Yaskawa INFORM job: pointsmerc3TRJ0.JBI

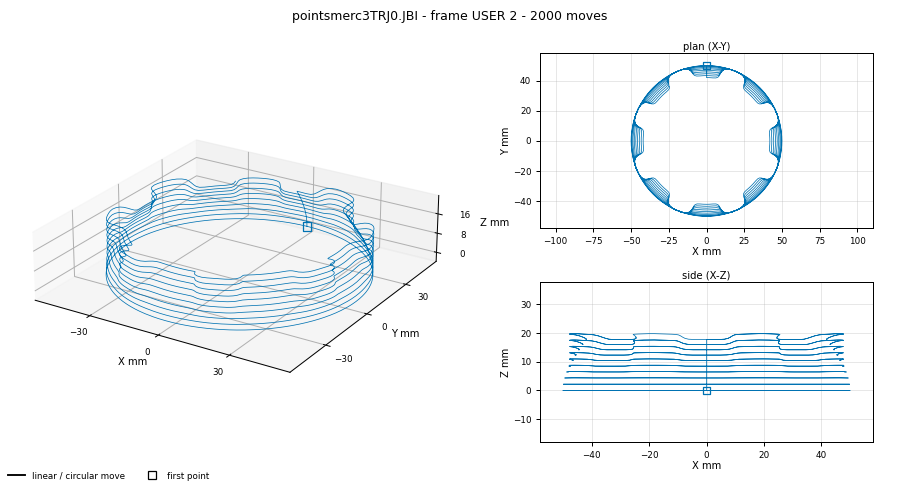
[picture p0: tool path of pointsmerc3TRJ0.JBI in frame USER 2, 2000 of 2000 moves have a stored position in this frame; points joined in program order, loops and branches not executed]
/JOB
//NAME pointsmerc3TRJ0
//POS
///NPOS 2000,0,0,0,0,0
///USER 2
///TOOL 1
///POSTYPE USER
///RECTAN
///RCONF 1,0,0,0,0,0,0,0,0,0,0,0,0,0,0,0,0,0,0,0,0,0,0,0
C00000=0.000,50.000,0.000,-180.0000,0.0000,0.0000
C00001=2.896,49.916,0.000,-180.0000,-0.0000,0.0000
C00002=5.494,49.697,0.000,-180.0000,-0.0000,0.0000
C00003=7.782,49.391,0.000,-180.0000,-0.0000,0.0000
C00004=9.349,49.118,0.000,-180.0000,-0.0000,0.0000
C00005=10.427,48.901,0.000,-180.0000,-0.0000,0.0000
C00006=11.297,48.707,0.000,-180.0000,-0.0000,0.0000
C00007=12.176,48.495,0.000,-180.0000,-0.0000,0.0000
C00008=13.275,48.206,0.000,-180.0000,-0.0000,0.0000
C00009=14.624,47.814,0.000,-180.0000,-0.0000,0.0000
C00010=16.047,47.355,0.000,-180.0000,-0.0000,0.0000
C00011=17.369,46.886,0.000,-180.0000,-0.0000,0.0000
C00012=18.561,46.427,0.000,-180.0000,-0.0000,0.0000
C00013=19.705,45.953,0.000,-180.0000,-0.0000,0.0000
C00014=20.871,45.435,0.000,-180.0000,-0.0000,0.0000
C00015=22.138,44.832,0.000,180.0000,0.0000,0.0000
C00016=23.469,44.150,0.000,180.0000,0.0000,0.0000
C00017=24.700,43.473,0.000,-180.0000,-0.0000,0.0000
C00018=25.682,42.901,0.000,-180.0000,-0.0000,0.0000
C00019=26.453,42.429,0.000,-180.0000,-0.0000,0.0000
C00020=27.205,41.951,0.000,-180.0000,-0.0000,0.0000
C00021=28.121,41.343,0.000,-180.0000,-0.0000,0.0000
C00022=29.422,40.427,0.000,-180.0000,-0.0000,0.0000
C00023=31.256,39.026,0.000,-180.0000,-0.0000,0.0000
C00024=33.248,37.344,0.000,-180.0000,-0.0000,0.0000
C00025=35.355,35.355,0.000,-180.0000,-0.0000,0.0000
C00026=37.344,33.248,0.000,-180.0000,-0.0000,0.0000
C00027=39.026,31.256,0.000,-180.0000,-0.0000,0.0000
C00028=40.427,29.422,0.000,180.0000,0.0000,0.0000
C00029=41.343,28.121,0.000,-180.0000,-0.0000,0.0000
C00030=41.951,27.205,0.000,-180.0000,-0.0000,0.0000
C00031=42.429,26.453,0.000,-180.0000,-0.0000,0.0000
C00032=42.901,25.682,0.000,-180.0000,-0.0000,0.0000
C00033=43.473,24.700,0.000,-180.0000,-0.0000,0.0000
C00034=44.150,23.469,0.000,-180.0000,-0.0000,0.0000
C00035=44.832,22.138,0.000,-180.0000,-0.0000,0.0000
C00036=45.435,20.871,0.000,-180.0000,-0.0000,0.0000
C00037=45.953,19.705,0.000,-180.0000,-0.0000,0.0000
C00038=46.427,18.561,0.000,-180.0000,-0.0000,0.0000
C00039=46.886,17.369,0.000,-180.0000,-0.0000,0.0000
C00040=47.355,16.047,0.000,-180.0000,-0.0000,0.0000
C00041=47.814,14.624,0.000,-180.0000,-0.0000,0.0000
C00042=48.206,13.275,0.000,-180.0000,-0.0000,0.0000
C00043=48.495,12.176,0.000,-180.0000,-0.0000,0.0000
C00044=48.707,11.297,0.000,-180.0000,-0.0000,0.0000
C00045=48.901,10.427,0.000,-180.0000,-0.0000,0.0000
C00046=49.118,9.349,0.000,-180.0000,-0.0000,0.0000
C00047=49.391,7.782,0.000,-180.0000,-0.0000,0.0000
C00048=49.697,5.494,0.000,-180.0000,-0.0000,0.0000
C00049=49.916,2.896,0.000,-180.0000,-0.0000,0.0000
C00050=50.000,0.000,0.000,-180.0000,-0.0000,0.0000
C00051=49.916,-2.896,0.000,180.0000,-0.0000,0.0000
C00052=49.697,-5.494,0.000,180.0000,-0.0000,0.0000
C00053=49.391,-7.782,0.000,180.0000,-0.0000,0.0000
C00054=49.118,-9.349,0.000,180.0000,-0.0000,0.0000
C00055=48.901,-10.427,0.000,180.0000,-0.0000,0.0000
C00056=48.707,-11.297,0.000,180.0000,-0.0000,0.0000
C00057=48.495,-12.176,0.000,180.0000,-0.0000,0.0000
C00058=48.206,-13.275,0.000,180.0000,-0.0000,0.0000
C00059=47.814,-14.624,0.000,180.0000,-0.0000,0.0000
C00060=47.355,-16.047,0.000,180.0000,-0.0000,0.0000
C00061=46.886,-17.369,0.000,180.0000,-0.0000,0.0000
C00062=46.427,-18.561,0.000,180.0000,-0.0000,0.0000
C00063=45.953,-19.705,0.000,180.0000,-0.0000,0.0000
C00064=45.435,-20.871,0.000,180.0000,-0.0000,0.0000
C00065=44.832,-22.138,0.000,180.0000,-0.0000,0.0000
C00066=44.150,-23.469,0.000,180.0000,-0.0000,0.0000
C00067=43.473,-24.700,0.000,180.0000,-0.0000,0.0000
C00068=42.901,-25.682,0.000,180.0000,-0.0000,0.0000
C00069=42.429,-26.453,0.000,180.0000,-0.0000,0.0000
C00070=41.951,-27.205,0.000,180.0000,-0.0000,0.0000
C00071=41.343,-28.121,0.000,180.0000,-0.0000,0.0000
C00072=40.427,-29.422,0.000,180.0000,-0.0000,0.0000
C00073=39.026,-31.256,0.000,180.0000,-0.0000,0.0000
C00074=37.344,-33.248,0.000,180.0000,-0.0000,0.0000
C00075=35.355,-35.355,0.000,180.0000,-0.0000,0.0000
C00076=33.248,-37.344,0.000,180.0000,-0.0000,0.0000
C00077=31.256,-39.026,0.000,180.0000,-0.0000,0.0000
C00078=29.422,-40.427,0.000,180.0000,-0.0000,0.0000
C00079=28.121,-41.343,0.000,180.0000,-0.0000,0.0000
C00080=27.205,-41.951,0.000,180.0000,-0.0000,0.0000
C00081=26.453,-42.429,0.000,180.0000,-0.0000,0.0000
C00082=25.682,-42.901,0.000,180.0000,-0.0000,0.0000
C00083=24.700,-43.473,0.000,-180.0000,0.0000,0.0000
C00084=23.469,-44.150,0.000,180.0000,-0.0000,0.0000
C00085=22.138,-44.832,0.000,180.0000,-0.0000,0.0000
C00086=20.871,-45.435,0.000,180.0000,-0.0000,0.0000
C00087=19.705,-45.953,0.000,180.0000,-0.0000,0.0000
C00088=18.561,-46.427,0.000,180.0000,-0.0000,0.0000
C00089=17.369,-46.886,0.000,180.0000,-0.0000,0.0000
C00090=16.047,-47.355,0.000,180.0000,-0.0000,0.0000
C00091=14.624,-47.814,0.000,180.0000,-0.0000,0.0000
C00092=13.275,-48.206,0.000,180.0000,-0.0000,0.0000
C00093=12.176,-48.495,0.000,180.0000,-0.0000,0.0000
C00094=11.297,-48.707,0.000,180.0000,-0.0000,0.0000
C00095=10.427,-48.901,0.000,180.0000,-0.0000,0.0000
C00096=9.349,-49.118,0.000,180.0000,-0.0000,0.0000
C00097=7.782,-49.391,0.000,180.0000,-0.0000,0.0000
C00098=5.494,-49.697,0.000,180.0000,-0.0000,0.0000
C00099=2.896,-49.916,0.000,180.0000,-0.0000,0.0000
C00100=0.000,-50.000,0.000,-180.0000,-0.0000,0.0000
C00101=0.000,-50.000,0.000,-180.0000,-0.0000,0.0000
C00102=-2.896,-49.916,0.000,-180.0000,-0.0000,0.0000
C00103=-5.494,-49.697,0.000,-180.0000,-0.0000,0.0000
C00104=-7.782,-49.391,0.000,-180.0000,-0.0000,0.0000
C00105=-9.349,-49.118,0.000,-180.0000,-0.0000,0.0000
C00106=-10.427,-48.901,0.000,-180.0000,-0.0000,0.0000
C00107=-11.297,-48.707,0.000,-180.0000,-0.0000,0.0000
C00108=-12.176,-48.495,0.000,-180.0000,-0.0000,0.0000
C00109=-13.275,-48.206,0.000,-180.0000,-0.0000,0.0000
C00110=-14.624,-47.814,0.000,-180.0000,-0.0000,0.0000
C00111=-16.047,-47.355,0.000,-180.0000,-0.0000,0.0000
C00112=-17.369,-46.886,0.000,-180.0000,-0.0000,0.0000
C00113=-18.561,-46.427,0.000,-180.0000,-0.0000,0.0000
C00114=-19.705,-45.953,0.000,-180.0000,-0.0000,0.0000
C00115=-20.871,-45.435,0.000,-180.0000,-0.0000,0.0000
C00116=-22.138,-44.832,0.000,-180.0000,-0.0000,0.0000
C00117=-23.469,-44.150,0.000,-180.0000,-0.0000,0.0000
C00118=-24.700,-43.473,0.000,-180.0000,-0.0000,0.0000
C00119=-25.682,-42.901,0.000,-180.0000,-0.0000,0.0000
C00120=-26.453,-42.429,0.000,-180.0000,-0.0000,0.0000
C00121=-27.205,-41.951,0.000,-180.0000,-0.0000,0.0000
C00122=-28.121,-41.343,0.000,-180.0000,-0.0000,0.0000
C00123=-29.422,-40.427,0.000,-180.0000,-0.0000,0.0000
C00124=-31.256,-39.026,0.000,-180.0000,-0.0000,0.0000
C00125=-33.248,-37.344,0.000,-180.0000,-0.0000,0.0000
C00126=-35.355,-35.355,0.000,-180.0000,-0.0000,0.0000
C00127=-37.344,-33.248,0.000,-180.0000,-0.0000,0.0000
C00128=-39.026,-31.256,0.000,-180.0000,-0.0000,0.0000
C00129=-40.427,-29.422,0.000,-180.0000,-0.0000,0.0000
C00130=-41.343,-28.121,0.000,-180.0000,-0.0000,0.0000
C00131=-41.951,-27.205,0.000,-180.0000,-0.0000,0.0000
C00132=-42.429,-26.453,0.000,-180.0000,-0.0000,0.0000
C00133=-42.901,-25.682,0.000,-180.0000,-0.0000,0.0000
C00134=-43.473,-24.700,0.000,-180.0000,-0.0000,0.0000
C00135=-44.150,-23.469,0.000,-180.0000,-0.0000,0.0000
C00136=-44.832,-22.138,0.000,-180.0000,-0.0000,0.0000
C00137=-45.435,-20.871,0.000,180.0000,0.0000,0.0000
C00138=-45.953,-19.705,0.000,180.0000,0.0000,0.0000
C00139=-46.427,-18.561,0.000,-180.0000,-0.0000,0.0000
C00140=-46.886,-17.369,0.000,-180.0000,-0.0000,0.0000
C00141=-47.355,-16.047,0.000,180.0000,0.0000,0.0000
C00142=-47.814,-14.624,0.000,180.0000,0.0000,0.0000
C00143=-48.206,-13.275,0.000,-180.0000,-0.0000,0.0000
C00144=-48.495,-12.176,0.000,-180.0000,-0.0000,0.0000
C00145=-48.707,-11.297,0.000,-180.0000,-0.0000,0.0000
C00146=-48.901,-10.427,0.000,-180.0000,-0.0000,0.0000
C00147=-49.118,-9.349,0.000,-180.0000,-0.0000,0.0000
C00148=-49.391,-7.782,0.000,-180.0000,-0.0000,0.0000
C00149=-49.697,-5.494,0.000,-180.0000,-0.0000,0.0000
C00150=-49.916,-2.896,0.000,-180.0000,-0.0000,0.0000
C00151=-50.000,0.000,0.000,180.0000,0.0000,0.0000
C00152=-49.916,2.896,0.000,-180.0000,0.0000,0.0000
C00153=-49.697,5.494,0.000,-180.0000,0.0000,0.0000
C00154=-49.391,7.782,0.000,-180.0000,0.0000,0.0000
C00155=-49.118,9.349,0.000,-180.0000,0.0000,0.0000
C00156=-48.901,10.427,0.000,-180.0000,0.0000,0.0000
C00157=-48.707,11.297,0.000,-180.0000,0.0000,0.0000
C00158=-48.495,12.176,0.000,-180.0000,0.0000,0.0000
C00159=-48.206,13.275,0.000,-180.0000,0.0000,0.0000
C00160=-47.814,14.624,0.000,-180.0000,0.0000,0.0000
C00161=-47.355,16.047,0.000,-180.0000,0.0000,0.0000
C00162=-46.886,17.369,0.000,-180.0000,0.0000,0.0000
C00163=-46.427,18.561,0.000,-180.0000,0.0000,0.0000
C00164=-45.953,19.705,0.000,-180.0000,0.0000,0.0000
C00165=-45.435,20.871,0.000,-180.0000,0.0000,0.0000
C00166=-44.832,22.138,0.000,-180.0000,0.0000,0.0000
C00167=-44.150,23.469,0.000,-180.0000,0.0000,0.0000
C00168=-43.473,24.700,0.000,-180.0000,0.0000,0.0000
C00169=-42.901,25.682,0.000,-180.0000,0.0000,0.0000
C00170=-42.429,26.453,0.000,-180.0000,0.0000,0.0000
C00171=-41.951,27.205,0.000,-180.0000,0.0000,0.0000
C00172=-41.343,28.121,0.000,-180.0000,0.0000,0.0000
C00173=-40.427,29.422,0.000,-180.0000,0.0000,0.0000
C00174=-39.026,31.256,0.000,-180.0000,0.0000,0.0000
C00175=-37.344,33.248,0.000,-180.0000,0.0000,0.0000
C00176=-35.355,35.355,0.000,-180.0000,0.0000,0.0000
C00177=-33.248,37.344,0.000,-180.0000,0.0000,0.0000
C00178=-31.256,39.026,0.000,-180.0000,0.0000,0.0000
C00179=-29.422,40.427,0.000,-180.0000,0.0000,0.0000
C00180=-28.121,41.343,0.000,-180.0000,0.0000,0.0000
C00181=-27.205,41.951,0.000,-180.0000,0.0000,0.0000
C00182=-26.453,42.429,0.000,-180.0000,0.0000,0.0000
C00183=-25.682,42.901,0.000,-180.0000,0.0000,0.0000
C00184=-24.700,43.473,0.000,-180.0000,0.0000,0.0000
C00185=-23.469,44.150,0.000,-180.0000,0.0000,0.0000
C00186=-22.138,44.832,0.000,-180.0000,0.0000,0.0000
C00187=-20.871,45.435,0.000,-180.0000,0.0000,0.0000
C00188=-19.705,45.953,0.000,-180.0000,0.0000,0.0000
C00189=-18.561,46.427,0.000,-180.0000,0.0000,0.0000
C00190=-17.369,46.886,0.000,-180.0000,0.0000,0.0000
C00191=-16.047,47.355,0.000,-180.0000,0.0000,0.0000
C00192=-14.624,47.814,0.000,-180.0000,0.0000,0.0000
C00193=-13.275,48.206,0.000,-180.0000,0.0000,0.0000
C00194=-12.176,48.495,0.000,-180.0000,0.0000,0.0000
C00195=-11.297,48.707,0.000,-180.0000,0.0000,0.0000
C00196=-10.427,48.901,0.000,-180.0000,0.0000,0.0000
C00197=-9.349,49.118,0.000,-180.0000,0.0000,0.0000
C00198=-7.782,49.391,0.000,-180.0000,0.0000,0.0000
C00199=-5.494,49.697,0.000,-180.0000,0.0000,0.0000
C00200=-2.896,49.916,0.000,-180.0000,0.0000,0.0000
C00201=0.000,50.000,0.000,-180.0000,0.0000,0.0000
C00202=0.000,49.846,2.195,-172.0982,0.0000,0.0000
C00203=2.882,49.762,2.195,-172.1070,-0.4575,0.0000
C00204=5.471,49.545,2.195,-172.1568,-0.8569,0.0000
C00205=7.753,49.245,2.195,-172.4939,-1.1371,0.0000
C00206=9.315,48.989,2.196,-173.2907,-1.1672,0.0000
C00207=10.389,48.795,2.197,-174.4353,-1.0311,0.0000
C00208=11.257,48.629,2.198,-175.7747,-0.8368,0.0000
C00209=12.134,48.445,2.199,-177.1182,-0.6422,0.0000
C00210=13.230,48.181,2.199,-178.2685,-0.4456,0.0000
C00211=14.582,47.809,2.200,-179.1783,-0.2412,0.0000
C00212=16.014,47.361,2.200,-179.7705,-0.0761,0.0000
C00213=17.348,46.893,2.200,-179.9632,-0.0136,0.0000
C00214=18.554,46.430,2.200,-179.9957,-0.0017,0.0000
C00215=19.712,45.950,2.200,-179.9957,-0.0018,0.0000
C00216=20.891,45.426,2.200,-179.9644,-0.0164,0.0000
C00217=22.166,44.813,2.200,-179.7839,-0.1085,0.0000
C00218=23.495,44.117,2.200,-179.2484,-0.4105,0.0000
C00219=24.714,43.424,2.199,-178.4604,-0.9091,0.0000
C00220=25.676,42.836,2.199,-177.5075,-1.5829,0.0000
C00221=26.426,42.346,2.198,-176.4182,-2.3937,0.0000
C00222=27.157,41.850,2.197,-175.3305,-3.2006,0.0000
C00223=28.054,41.227,2.196,-174.4206,-3.9102,0.0000
C00224=29.339,40.304,2.195,-173.8741,-4.4920,0.0000
C00225=31.165,38.902,2.195,-173.8314,-4.9282,0.0000
C00226=33.149,37.225,2.195,-174.0778,-5.2472,0.0000
C00227=35.246,35.246,2.195,-174.3948,-5.5785,0.0000
C00228=37.225,33.149,2.195,-174.7249,-5.8973,0.0000
C00229=38.902,31.165,2.195,-175.0432,-6.1458,0.0000
C00230=40.304,29.339,2.195,-175.4823,-6.1070,0.0000
C00231=41.227,28.054,2.196,-176.0713,-5.5664,0.0000
C00232=41.850,27.157,2.197,-176.7887,-4.6622,0.0000
C00233=42.346,26.426,2.198,-177.6016,-3.5787,0.0000
C00234=42.836,25.676,2.199,-178.4156,-2.4916,0.0000
C00235=43.424,24.714,2.199,-179.0906,-1.5394,0.0000
C00236=44.117,23.495,2.200,-179.5895,-0.7516,0.0000
C00237=44.813,22.166,2.200,-179.8915,-0.2161,0.0000
C00238=45.426,20.891,2.200,-179.9836,-0.0356,0.0000
C00239=45.950,19.712,2.200,-179.9982,-0.0043,0.0000
C00240=46.430,18.554,2.200,-179.9983,-0.0043,0.0000
C00241=46.893,17.348,2.200,-179.9864,-0.0368,0.0000
C00242=47.361,16.014,2.200,-179.9239,-0.2295,0.0000
C00243=47.809,14.582,2.200,-179.7588,-0.8217,0.0000
C00244=48.181,13.230,2.199,-179.5542,-1.7314,0.0000
C00245=48.445,12.134,2.199,-179.3570,-2.8816,0.0000
C00246=48.629,11.257,2.198,-179.1609,-4.2248,0.0000
C00247=48.795,10.389,2.197,-178.9640,-5.5638,0.0000
C00248=48.989,9.315,2.196,-178.8248,-6.7079,0.0000
C00249=49.245,7.753,2.195,-178.8530,-7.5046,0.0000
C00250=49.545,5.471,2.195,-179.1350,-7.8423,0.0000
C00251=49.762,2.882,2.195,-179.5381,-7.8927,0.0000
C00252=49.846,0.000,2.195,180.0000,-7.9018,0.0000
C00253=49.762,-2.882,2.195,179.5381,-7.8927,0.0000
C00254=49.545,-5.471,2.195,179.1350,-7.8423,0.0000
C00255=49.245,-7.753,2.195,178.8530,-7.5046,0.0000
C00256=48.989,-9.315,2.196,178.8248,-6.7079,0.0000
C00257=48.795,-10.389,2.197,178.9640,-5.5638,0.0000
C00258=48.629,-11.257,2.198,179.1609,-4.2248,0.0000
C00259=48.445,-12.134,2.199,179.3570,-2.8816,0.0000
C00260=48.181,-13.230,2.199,179.5542,-1.7314,0.0000
C00261=47.809,-14.582,2.200,179.7588,-0.8217,0.0000
C00262=47.361,-16.014,2.200,179.9239,-0.2295,0.0000
C00263=46.893,-17.348,2.200,179.9864,-0.0368,0.0000
C00264=46.430,-18.554,2.200,179.9983,-0.0043,0.0000
C00265=45.950,-19.712,2.200,179.9982,-0.0043,0.0000
C00266=45.426,-20.891,2.200,179.9836,-0.0356,0.0000
C00267=44.813,-22.166,2.200,179.8915,-0.2161,0.0000
C00268=44.117,-23.495,2.200,179.5895,-0.7516,0.0000
C00269=43.424,-24.714,2.199,179.0906,-1.5394,0.0000
C00270=42.836,-25.676,2.199,178.4156,-2.4916,0.0000
C00271=42.346,-26.426,2.198,177.6016,-3.5787,0.0000
C00272=41.850,-27.157,2.197,176.7887,-4.6622,0.0000
C00273=41.227,-28.054,2.196,176.0713,-5.5664,0.0000
C00274=40.304,-29.339,2.195,175.4823,-6.1070,0.0000
C00275=38.902,-31.165,2.195,175.0432,-6.1457,0.0000
C00276=37.225,-33.149,2.195,174.7248,-5.8973,0.0000
C00277=35.246,-35.246,2.195,174.3948,-5.5785,0.0000
C00278=33.149,-37.225,2.195,174.0778,-5.2471,0.0000
C00279=31.165,-38.902,2.195,173.8314,-4.9283,0.0000
C00280=29.339,-40.304,2.195,173.8742,-4.4920,0.0000
C00281=28.054,-41.227,2.196,174.4206,-3.9102,0.0000
C00282=27.157,-41.850,2.197,175.3305,-3.2006,0.0000
C00283=26.426,-42.346,2.198,176.4182,-2.3937,0.0000
C00284=25.676,-42.836,2.199,177.5075,-1.5829,0.0000
C00285=24.714,-43.424,2.199,178.4604,-0.9091,0.0000
C00286=23.495,-44.117,2.200,179.2484,-0.4105,0.0000
C00287=22.166,-44.813,2.200,179.7839,-0.1085,0.0000
C00288=20.891,-45.426,2.200,179.9644,-0.0164,0.0000
C00289=19.712,-45.950,2.200,179.9957,-0.0018,0.0000
C00290=18.554,-46.430,2.200,179.9957,-0.0017,0.0000
C00291=17.348,-46.893,2.200,179.9632,-0.0136,0.0000
C00292=16.014,-47.361,2.200,179.7705,-0.0761,0.0000
C00293=14.582,-47.809,2.200,179.1783,-0.2412,0.0000
C00294=13.230,-48.181,2.199,178.2685,-0.4456,0.0000
C00295=12.134,-48.445,2.199,177.1182,-0.6422,0.0000
C00296=11.257,-48.629,2.198,175.7747,-0.8368,0.0000
C00297=10.389,-48.795,2.197,174.4353,-1.0311,0.0000
C00298=9.315,-48.989,2.196,173.2907,-1.1672,0.0000
C00299=7.753,-49.245,2.195,172.4939,-1.1371,0.0000
C00300=5.471,-49.545,2.195,172.1568,-0.8569,0.0000
C00301=2.882,-49.762,2.195,172.1070,-0.4575,0.0000
C00302=0.000,-49.846,2.195,172.0982,0.0000,0.0000
C00303=0.000,-49.846,2.195,172.0982,0.0000,0.0000
C00304=-2.882,-49.762,2.195,172.1071,0.4575,0.0000
C00305=-5.471,-49.545,2.195,172.1568,0.8569,0.0000
C00306=-7.753,-49.245,2.195,172.4939,1.1371,0.0000
C00307=-9.315,-48.989,2.196,173.2907,1.1672,0.0000
C00308=-10.389,-48.795,2.197,174.4353,1.0311,0.0000
C00309=-11.257,-48.629,2.198,175.7747,0.8368,0.0000
C00310=-12.134,-48.445,2.199,177.1182,0.6422,0.0000
C00311=-13.230,-48.181,2.199,178.2685,0.4456,0.0000
C00312=-14.582,-47.809,2.200,179.1783,0.2412,0.0000
C00313=-16.014,-47.361,2.200,179.7705,0.0761,0.0000
C00314=-17.348,-46.893,2.200,179.9632,0.0136,0.0000
C00315=-18.554,-46.430,2.200,179.9957,0.0017,0.0000
C00316=-19.712,-45.950,2.200,179.9957,0.0018,0.0000
C00317=-20.891,-45.426,2.200,179.9644,0.0164,0.0000
C00318=-22.166,-44.813,2.200,179.7839,0.1085,0.0000
C00319=-23.495,-44.117,2.200,179.2484,0.4105,0.0000
C00320=-24.714,-43.424,2.199,178.4604,0.9091,0.0000
C00321=-25.676,-42.836,2.199,177.5075,1.5829,0.0000
C00322=-26.426,-42.346,2.198,176.4182,2.3937,0.0000
C00323=-27.157,-41.850,2.197,175.3305,3.2006,0.0000
C00324=-28.054,-41.227,2.196,174.4206,3.9102,0.0000
C00325=-29.339,-40.304,2.195,173.8741,4.4920,0.0000
C00326=-31.165,-38.902,2.195,173.8314,4.9282,0.0000
C00327=-33.149,-37.225,2.195,174.0778,5.2472,0.0000
C00328=-35.246,-35.246,2.195,174.3948,5.5785,0.0000
C00329=-37.225,-33.149,2.195,174.7249,5.8973,0.0000
C00330=-38.902,-31.165,2.195,175.0432,6.1458,0.0000
C00331=-40.304,-29.339,2.195,175.4823,6.1070,0.0000
C00332=-41.227,-28.054,2.196,176.0713,5.5664,0.0000
C00333=-41.850,-27.157,2.197,176.7887,4.6622,0.0000
C00334=-42.346,-26.426,2.198,177.6016,3.5787,0.0000
C00335=-42.836,-25.676,2.199,178.4156,2.4916,0.0000
C00336=-43.424,-24.714,2.199,179.0906,1.5394,0.0000
C00337=-44.117,-23.495,2.200,179.5895,0.7516,0.0000
C00338=-44.813,-22.166,2.200,179.8915,0.2161,0.0000
C00339=-45.426,-20.891,2.200,179.9836,0.0356,0.0000
C00340=-45.950,-19.712,2.200,179.9982,0.0043,0.0000
C00341=-46.430,-18.554,2.200,179.9983,0.0043,0.0000
C00342=-46.893,-17.348,2.200,179.9864,0.0368,0.0000
C00343=-47.361,-16.014,2.200,179.9239,0.2295,0.0000
C00344=-47.809,-14.582,2.200,179.7588,0.8217,0.0000
C00345=-48.181,-13.230,2.199,179.5542,1.7314,0.0000
C00346=-48.445,-12.134,2.199,179.3570,2.8816,0.0000
C00347=-48.629,-11.257,2.198,179.1609,4.2248,0.0000
C00348=-48.795,-10.389,2.197,178.9640,5.5638,0.0000
C00349=-48.989,-9.315,2.196,178.8248,6.7079,0.0000
C00350=-49.245,-7.753,2.195,178.8530,7.5046,0.0000
C00351=-49.545,-5.471,2.195,179.1350,7.8423,0.0000
C00352=-49.762,-2.882,2.195,179.5381,7.8927,0.0000
C00353=-49.846,0.000,2.195,-180.0000,7.9018,0.0000
C00354=-49.762,2.882,2.195,-179.5381,7.8927,0.0000
C00355=-49.545,5.471,2.195,-179.1350,7.8423,0.0000
C00356=-49.245,7.753,2.195,-178.8530,7.5046,0.0000
C00357=-48.989,9.315,2.196,-178.8248,6.7079,0.0000
C00358=-48.795,10.389,2.197,-178.9640,5.5638,0.0000
C00359=-48.629,11.257,2.198,-179.1609,4.2248,0.0000
C00360=-48.445,12.134,2.199,-179.3570,2.8816,0.0000
C00361=-48.181,13.230,2.199,-179.5542,1.7314,0.0000
C00362=-47.809,14.582,2.200,-179.7588,0.8217,0.0000
C00363=-47.361,16.014,2.200,-179.9239,0.2295,0.0000
C00364=-46.893,17.348,2.200,-179.9864,0.0368,0.0000
C00365=-46.430,18.554,2.200,-179.9983,0.0043,0.0000
C00366=-45.950,19.712,2.200,-179.9982,0.0043,0.0000
C00367=-45.426,20.891,2.200,-179.9836,0.0356,0.0000
C00368=-44.813,22.166,2.200,-179.8915,0.2161,0.0000
C00369=-44.117,23.495,2.200,-179.5895,0.7516,0.0000
C00370=-43.424,24.714,2.199,-179.0906,1.5394,0.0000
C00371=-42.836,25.676,2.199,-178.4156,2.4916,0.0000
C00372=-42.346,26.426,2.198,-177.6016,3.5787,0.0000
C00373=-41.850,27.157,2.197,-176.7887,4.6622,0.0000
C00374=-41.227,28.054,2.196,-176.0713,5.5664,0.0000
C00375=-40.304,29.339,2.195,-175.4823,6.1070,0.0000
C00376=-38.902,31.165,2.195,-175.0432,6.1457,0.0000
C00377=-37.225,33.149,2.195,-174.7248,5.8973,0.0000
C00378=-35.246,35.246,2.195,-174.3948,5.5785,0.0000
C00379=-33.149,37.225,2.195,-174.0778,5.2471,0.0000
C00380=-31.165,38.902,2.195,-173.8314,4.9283,0.0000
C00381=-29.339,40.304,2.195,-173.8742,4.4920,0.0000
C00382=-28.054,41.227,2.196,-174.4206,3.9102,0.0000
C00383=-27.157,41.850,2.197,-175.3305,3.2006,0.0000
C00384=-26.426,42.346,2.198,-176.4182,2.3937,0.0000
C00385=-25.676,42.836,2.199,-177.5075,1.5829,0.0000
C00386=-24.714,43.424,2.199,-178.4604,0.9091,0.0000
C00387=-23.495,44.117,2.200,-179.2484,0.4105,0.0000
C00388=-22.166,44.813,2.200,-179.7839,0.1085,0.0000
C00389=-20.891,45.426,2.200,-179.9644,0.0164,0.0000
C00390=-19.712,45.950,2.200,-179.9957,0.0018,0.0000
C00391=-18.554,46.430,2.200,-179.9957,0.0017,0.0000
C00392=-17.348,46.893,2.200,-179.9632,0.0136,0.0000
C00393=-16.014,47.361,2.200,-179.7705,0.0761,0.0000
C00394=-14.582,47.809,2.200,-179.1783,0.2412,0.0000
C00395=-13.230,48.181,2.199,-178.2685,0.4456,0.0000
C00396=-12.134,48.445,2.199,-177.1182,0.6422,0.0000
C00397=-11.257,48.629,2.198,-175.7747,0.8368,0.0000
C00398=-10.389,48.795,2.197,-174.4353,1.0311,0.0000
C00399=-9.315,48.989,2.196,-173.2907,1.1672,0.0000
C00400=-7.753,49.245,2.195,-172.4939,1.1371,0.0000
C00401=-5.471,49.545,2.195,-172.1568,0.8569,0.0000
C00402=-2.882,49.762,2.195,-172.1071,0.4575,0.0000
C00403=0.000,49.846,2.195,-172.0982,0.0000,0.0000
C00404=0.000,49.410,4.351,-165.2330,0.0000,0.0000
C00405=2.842,49.327,4.351,-165.2490,-0.8462,0.0000
C00406=5.404,49.114,4.351,-165.3368,-1.5509,0.0000
C00407=7.672,48.833,4.355,-165.9287,-1.8917,0.0000
C00408=9.218,48.623,4.363,-167.3753,-1.6057,0.0000
C00409=10.282,48.495,4.374,-169.5506,-1.1016,0.0000
C00410=11.143,48.407,4.384,-172.1383,-0.7944,0.0000
C00411=12.014,48.303,4.391,-174.6908,-0.7528,0.0000
C00412=13.101,48.111,4.395,-176.8484,-0.6476,0.0000
C00413=14.461,47.794,4.396,-178.5414,-0.3774,0.0000
C00414=15.918,47.378,4.398,-179.6165,-0.1196,0.0000
C00415=17.289,46.913,4.399,-179.9364,-0.0233,0.0000
C00416=18.533,46.438,4.400,-179.9926,-0.0029,0.0000
C00417=19.732,45.942,4.400,-179.9927,-0.0031,0.0000
C00418=20.948,45.397,4.399,-179.9386,-0.0286,0.0000
C00419=22.246,44.758,4.398,-179.6442,-0.1866,0.0000
C00420=23.570,44.021,4.396,-178.7016,-0.7644,0.0000
C00421=24.756,43.284,4.395,-177.3126,-1.7696,0.0000
C00422=25.660,42.651,4.391,-175.7085,-3.2179,0.0000
C00423=26.350,42.108,4.384,-173.8623,-4.9857,0.0000
C00424=27.021,41.562,4.374,-171.7926,-6.5822,0.0000
C00425=27.864,40.900,4.363,-169.8688,-7.7398,0.0000
C00426=29.106,39.955,4.355,-168.6177,-8.5390,0.0000
C00427=30.908,38.550,4.351,-168.4253,-9.1948,0.0000
C00428=32.870,36.889,4.351,-168.8566,-9.7634,0.0000
C00429=34.938,34.938,4.351,-169.4418,-10.3834,0.0000
C00430=36.889,32.870,4.351,-170.0527,-10.9799,0.0000
C00431=38.550,30.908,4.351,-170.6177,-11.4240,0.0000
C00432=39.955,29.106,4.355,-171.2923,-11.2544,0.0000
C00433=40.900,27.864,4.363,-172.1392,-10.0380,0.0000
C00434=41.562,27.021,4.374,-173.3503,-8.1529,0.0000
C00435=42.108,26.350,4.384,-174.9857,-6.1144,0.0000
C00436=42.651,25.660,4.391,-176.7731,-4.2848,0.0000
C00437=43.284,24.756,4.395,-178.2285,-2.6861,0.0000
C00438=44.021,23.570,4.396,-179.2354,-1.2982,0.0000
C00439=44.758,22.246,4.398,-179.8134,-0.3558,0.0000
C00440=45.397,20.948,4.399,-179.9714,-0.0614,0.0000
C00441=45.942,19.732,4.400,-179.9969,-0.0073,0.0000
C00442=46.438,18.533,4.400,-179.9971,-0.0074,0.0000
C00443=46.913,17.289,4.399,-179.9767,-0.0636,0.0000
C00444=47.378,15.918,4.398,-179.8804,-0.3835,0.0000
C00445=47.794,14.461,4.396,-179.6224,-1.4586,0.0000
C00446=48.111,13.101,4.395,-179.3514,-3.1514,0.0000
C00447=48.303,12.014,4.391,-179.2440,-5.3088,0.0000
C00448=48.407,11.143,4.384,-179.1981,-7.8609,0.0000
C00449=48.495,10.282,4.374,-178.8799,-10.4474,0.0000
C00450=48.623,9.218,4.363,-178.3546,-12.6196,0.0000
C00451=48.833,7.672,4.355,-178.0498,-14.0635,0.0000
C00452=49.114,5.404,4.351,-178.3969,-14.6577,0.0000
C00453=49.327,2.842,4.351,-179.1250,-14.7494,0.0000
C00454=49.410,0.000,4.351,180.0000,-14.7670,0.0000
C00455=49.327,-2.842,4.351,179.1250,-14.7493,0.0000
C00456=49.114,-5.404,4.351,178.3969,-14.6578,0.0000
C00457=48.833,-7.672,4.355,178.0498,-14.0634,0.0000
C00458=48.623,-9.218,4.363,178.3546,-12.6196,0.0000
C00459=48.495,-10.282,4.374,178.8799,-10.4474,0.0000
C00460=48.407,-11.143,4.384,179.1981,-7.8609,0.0000
C00461=48.303,-12.014,4.391,179.2440,-5.3088,0.0000
C00462=48.111,-13.101,4.395,179.3514,-3.1514,0.0000
C00463=47.794,-14.461,4.396,179.6224,-1.4586,0.0000
C00464=47.378,-15.918,4.398,179.8804,-0.3835,0.0000
C00465=46.913,-17.289,4.399,179.9767,-0.0636,0.0000
C00466=46.438,-18.533,4.400,179.9971,-0.0074,0.0000
C00467=45.942,-19.732,4.400,179.9969,-0.0073,0.0000
C00468=45.397,-20.948,4.399,179.9714,-0.0614,0.0000
C00469=44.758,-22.246,4.398,179.8134,-0.3558,0.0000
C00470=44.021,-23.570,4.396,179.2354,-1.2982,0.0000
C00471=43.284,-24.756,4.395,178.2285,-2.6861,0.0000
C00472=42.651,-25.660,4.391,176.7731,-4.2848,0.0000
C00473=42.108,-26.350,4.384,174.9857,-6.1144,0.0000
C00474=41.562,-27.021,4.374,173.3503,-8.1529,0.0000
C00475=40.900,-27.864,4.363,172.1392,-10.0380,0.0000
C00476=39.955,-29.106,4.355,171.2923,-11.2544,0.0000
C00477=38.550,-30.908,4.351,170.6177,-11.4240,0.0000
C00478=36.889,-32.870,4.351,170.0527,-10.9800,0.0000
C00479=34.938,-34.938,4.351,169.4417,-10.3834,0.0000
C00480=32.870,-36.889,4.351,168.8567,-9.7634,0.0000
C00481=30.908,-38.550,4.351,168.4253,-9.1948,0.0000
C00482=29.106,-39.955,4.355,168.6177,-8.5390,0.0000
C00483=27.864,-40.900,4.363,169.8688,-7.7398,0.0000
C00484=27.021,-41.562,4.374,171.7926,-6.5822,0.0000
C00485=26.350,-42.108,4.384,173.8623,-4.9857,0.0000
C00486=25.660,-42.651,4.391,175.7085,-3.2179,0.0000
C00487=24.756,-43.284,4.395,177.3126,-1.7696,0.0000
C00488=23.570,-44.021,4.396,178.7016,-0.7644,0.0000
C00489=22.246,-44.758,4.398,179.6442,-0.1866,0.0000
C00490=20.948,-45.397,4.399,179.9386,-0.0286,0.0000
C00491=19.732,-45.942,4.400,179.9927,-0.0031,0.0000
C00492=18.533,-46.438,4.400,179.9926,-0.0029,0.0000
C00493=17.289,-46.913,4.399,179.9364,-0.0233,0.0000
C00494=15.918,-47.378,4.398,179.6165,-0.1196,0.0000
C00495=14.461,-47.794,4.396,178.5414,-0.3774,0.0000
C00496=13.101,-48.111,4.395,176.8484,-0.6476,0.0000
C00497=12.014,-48.303,4.391,174.6908,-0.7528,0.0000
C00498=11.143,-48.407,4.384,172.1383,-0.7944,0.0000
C00499=10.282,-48.495,4.374,169.5506,-1.1016,0.0000
C00500=9.218,-48.623,4.363,167.3753,-1.6057,0.0000
C00501=7.672,-48.833,4.355,165.9287,-1.8917,0.0000
C00502=5.404,-49.114,4.351,165.3368,-1.5509,0.0000
C00503=2.842,-49.327,4.351,165.2490,-0.8462,0.0000
C00504=0.000,-49.410,4.351,165.2330,0.0000,0.0000
C00505=0.000,-49.410,4.351,165.2330,0.0000,0.0000
C00506=-2.842,-49.327,4.351,165.2490,0.8461,0.0000
C00507=-5.404,-49.114,4.351,165.3367,1.5509,0.0000
C00508=-7.672,-48.833,4.355,165.9288,1.8917,0.0000
C00509=-9.218,-48.623,4.363,167.3753,1.6057,0.0000
C00510=-10.282,-48.495,4.374,169.5506,1.1016,0.0000
C00511=-11.143,-48.407,4.384,172.1383,0.7944,0.0000
C00512=-12.014,-48.303,4.391,174.6908,0.7528,0.0000
C00513=-13.101,-48.111,4.395,176.8484,0.6476,0.0000
C00514=-14.461,-47.794,4.396,178.5414,0.3774,0.0000
C00515=-15.918,-47.378,4.398,179.6165,0.1196,0.0000
C00516=-17.289,-46.913,4.399,179.9364,0.0233,0.0000
C00517=-18.533,-46.438,4.400,179.9926,0.0029,0.0000
C00518=-19.732,-45.942,4.400,179.9927,0.0031,0.0000
C00519=-20.948,-45.397,4.399,179.9386,0.0286,0.0000
C00520=-22.246,-44.758,4.398,179.6442,0.1866,0.0000
C00521=-23.570,-44.021,4.396,178.7016,0.7644,0.0000
C00522=-24.756,-43.284,4.395,177.3126,1.7696,0.0000
C00523=-25.660,-42.651,4.391,175.7085,3.2179,0.0000
C00524=-26.350,-42.108,4.384,173.8623,4.9857,0.0000
C00525=-27.021,-41.562,4.374,171.7926,6.5822,0.0000
C00526=-27.864,-40.900,4.363,169.8688,7.7398,0.0000
C00527=-29.106,-39.955,4.355,168.6177,8.5390,0.0000
C00528=-30.908,-38.550,4.351,168.4253,9.1948,0.0000
C00529=-32.870,-36.889,4.351,168.8566,9.7634,0.0000
C00530=-34.938,-34.938,4.351,169.4418,10.3834,0.0000
C00531=-36.889,-32.870,4.351,170.0527,10.9799,0.0000
C00532=-38.550,-30.908,4.351,170.6177,11.4240,0.0000
C00533=-39.955,-29.106,4.355,171.2923,11.2544,0.0000
C00534=-40.900,-27.864,4.363,172.1392,10.0380,0.0000
C00535=-41.562,-27.021,4.374,173.3503,8.1529,0.0000
C00536=-42.108,-26.350,4.384,174.9857,6.1144,0.0000
C00537=-42.651,-25.660,4.391,176.7731,4.2848,0.0000
C00538=-43.284,-24.756,4.395,178.2285,2.6861,0.0000
C00539=-44.021,-23.570,4.396,179.2354,1.2982,0.0000
C00540=-44.758,-22.246,4.398,179.8134,0.3558,0.0000
C00541=-45.397,-20.948,4.399,179.9714,0.0614,0.0000
C00542=-45.942,-19.732,4.400,179.9969,0.0073,0.0000
C00543=-46.438,-18.533,4.400,179.9971,0.0074,0.0000
C00544=-46.913,-17.289,4.399,179.9767,0.0636,0.0000
C00545=-47.378,-15.918,4.398,179.8804,0.3835,0.0000
C00546=-47.794,-14.461,4.396,179.6224,1.4586,0.0000
C00547=-48.111,-13.101,4.395,179.3514,3.1514,0.0000
C00548=-48.303,-12.014,4.391,179.2440,5.3088,0.0000
C00549=-48.407,-11.143,4.384,179.1981,7.8609,0.0000
C00550=-48.495,-10.282,4.374,178.8799,10.4474,0.0000
C00551=-48.623,-9.218,4.363,178.3546,12.6196,0.0000
C00552=-48.833,-7.672,4.355,178.0498,14.0635,0.0000
C00553=-49.114,-5.404,4.351,178.3969,14.6577,0.0000
C00554=-49.327,-2.842,4.351,179.1250,14.7494,0.0000
C00555=-49.410,0.000,4.351,-180.0000,14.7670,0.0000
C00556=-49.327,2.842,4.351,-179.1250,14.7493,0.0000
C00557=-49.114,5.404,4.351,-178.3969,14.6578,0.0000
C00558=-48.833,7.672,4.355,-178.0498,14.0634,0.0000
C00559=-48.623,9.218,4.363,-178.3546,12.6196,0.0000
C00560=-48.495,10.282,4.374,-178.8799,10.4474,0.0000
C00561=-48.407,11.143,4.384,-179.1981,7.8609,0.0000
C00562=-48.303,12.014,4.391,-179.2440,5.3088,0.0000
C00563=-48.111,13.101,4.395,-179.3514,3.1514,0.0000
C00564=-47.794,14.461,4.396,-179.6224,1.4586,0.0000
C00565=-47.378,15.918,4.398,-179.8804,0.3835,0.0000
C00566=-46.913,17.289,4.399,-179.9767,0.0636,0.0000
C00567=-46.438,18.533,4.400,-179.9971,0.0074,0.0000
C00568=-45.942,19.732,4.400,-179.9969,0.0073,0.0000
C00569=-45.397,20.948,4.399,-179.9714,0.0614,0.0000
C00570=-44.758,22.246,4.398,-179.8134,0.3558,0.0000
C00571=-44.021,23.570,4.396,-179.2354,1.2982,0.0000
C00572=-43.284,24.756,4.395,-178.2285,2.6861,0.0000
C00573=-42.651,25.660,4.391,-176.7731,4.2848,0.0000
C00574=-42.108,26.350,4.384,-174.9857,6.1144,0.0000
C00575=-41.562,27.021,4.374,-173.3503,8.1529,0.0000
C00576=-40.900,27.864,4.363,-172.1392,10.0380,0.0000
C00577=-39.955,29.106,4.355,-171.2923,11.2544,0.0000
C00578=-38.550,30.908,4.351,-170.6177,11.4240,0.0000
C00579=-36.889,32.870,4.351,-170.0527,10.9800,0.0000
C00580=-34.938,34.938,4.351,-169.4417,10.3834,0.0000
C00581=-32.870,36.889,4.351,-168.8567,9.7634,0.0000
C00582=-30.908,38.550,4.351,-168.4253,9.1948,0.0000
C00583=-29.106,39.955,4.355,-168.6177,8.5390,0.0000
C00584=-27.864,40.900,4.363,-169.8688,7.7398,0.0000
C00585=-27.021,41.562,4.374,-171.7926,6.5822,0.0000
C00586=-26.350,42.108,4.384,-173.8623,4.9857,0.0000
C00587=-25.660,42.651,4.391,-175.7085,3.2179,0.0000
C00588=-24.756,43.284,4.395,-177.3126,1.7696,0.0000
C00589=-23.570,44.021,4.396,-178.7016,0.7644,0.0000
C00590=-22.246,44.758,4.398,-179.6442,0.1866,0.0000
C00591=-20.948,45.397,4.399,-179.9386,0.0286,0.0000
C00592=-19.732,45.942,4.400,-179.9927,0.0031,0.0000
C00593=-18.533,46.438,4.400,-179.9926,0.0029,0.0000
C00594=-17.289,46.913,4.399,-179.9364,0.0233,0.0000
C00595=-15.918,47.378,4.398,-179.6165,0.1196,0.0000
C00596=-14.461,47.794,4.396,-178.5414,0.3774,0.0000
C00597=-13.101,48.111,4.395,-176.8484,0.6476,0.0000
C00598=-12.014,48.303,4.391,-174.6908,0.7528,0.0000
C00599=-11.143,48.407,4.384,-172.1383,0.7944,0.0000
C00600=-10.282,48.495,4.374,-169.5506,1.1016,0.0000
C00601=-9.218,48.623,4.363,-167.3753,1.6057,0.0000
C00602=-7.672,48.833,4.355,-165.9288,1.8917,0.0000
C00603=-5.404,49.114,4.351,-165.3367,1.5509,0.0000
C00604=-2.842,49.327,4.351,-165.2490,0.8461,0.0000
C00605=0.000,49.410,4.351,-165.2330,0.0000,0.0000
C00606=0.000,48.740,6.447,-159.5183,0.0001,0.0000
C00607=2.781,48.660,6.446,-159.5397,-1.1571,0.0000
C00608=5.301,48.453,6.447,-159.6520,-2.0469,0.0000
C00609=7.547,48.199,6.458,-160.4168,-2.1209,0.0000
C00610=9.067,48.057,6.484,-162.4669,-0.9364,0.0000
C00611=10.113,48.028,6.517,-165.7953,0.2947,0.0000
C00612=10.965,48.058,6.549,-169.6341,0.5477,0.0000
C00613=11.826,48.078,6.572,-173.0614,-0.0815,0.0000
C00614=12.898,48.000,6.582,-175.9035,-0.5039,0.0000
C00615=14.270,47.771,6.588,-178.1724,-0.3758,0.0000
C00616=15.768,47.406,6.592,-179.5717,-0.1209,0.0000
C00617=17.193,46.944,6.597,-179.9229,-0.0278,0.0000
C00618=18.501,46.450,6.600,-179.9912,-0.0035,0.0000
C00619=19.763,45.928,6.600,-179.9913,-0.0038,0.0000
C00620=21.037,45.352,6.597,-179.9258,-0.0349,0.0000
C00621=22.372,44.670,6.592,-179.6117,-0.2174,0.0000
C00622=23.689,43.870,6.588,-178.4417,-1.0264,0.0000
C00623=24.821,43.061,6.582,-176.7447,-2.5386,0.0000
C00624=25.634,42.359,6.572,-175.0240,-4.8425,0.0000
C00625=26.229,41.735,6.549,-173.0177,-7.7000,0.0000
C00626=26.810,41.112,6.517,-170.0607,-10.2038,0.0000
C00627=27.570,40.393,6.484,-166.7472,-11.6210,0.0000
C00628=28.746,39.419,6.458,-164.3922,-12.1618,0.0000
C00629=30.513,38.009,6.447,-163.8705,-12.7362,0.0000
C00630=32.441,36.374,6.446,-164.4076,-13.4647,0.0000
C00631=34.464,34.464,6.447,-165.2050,-14.3251,0.0000
C00632=36.374,32.441,6.446,-166.0406,-15.1532,0.0000
C00633=38.009,30.513,6.447,-166.7598,-15.7222,0.0000
C00634=39.419,28.746,6.458,-167.3873,-15.2489,0.0000
C00635=40.393,27.570,6.484,-168.0701,-12.9763,0.0000
C00636=41.112,26.810,6.517,-169.6441,-9.7806,0.0000
C00637=41.735,26.229,6.549,-172.2431,-6.9191,0.0000
C00638=42.359,25.634,6.572,-175.1392,-4.9582,0.0000
C00639=43.061,24.821,6.582,-177.4573,-3.2521,0.0000
C00640=43.870,23.689,6.588,-178.9732,-1.5580,0.0000
C00641=44.670,22.372,6.592,-179.7826,-0.3883,0.0000
C00642=45.352,21.037,6.597,-179.9651,-0.0742,0.0000
C00643=45.928,19.763,6.600,-179.9962,-0.0087,0.0000
C00644=46.450,18.501,6.600,-179.9965,-0.0088,0.0000
C00645=46.944,17.193,6.597,-179.9722,-0.0771,0.0000
C00646=47.406,15.768,6.592,-179.8791,-0.4283,0.0000
C00647=47.771,14.270,6.588,-179.6240,-1.8276,0.0000
C00648=48.000,12.898,6.582,-179.4948,-4.0963,0.0000
C00649=48.078,11.826,6.572,-179.9179,-6.9386,0.0000
C00650=48.058,10.965,6.549,179.4432,-10.3655,0.0000
C00651=48.028,10.113,6.517,179.6960,-14.2045,0.0000
C00652=48.057,9.067,6.484,-179.0180,-17.5307,0.0000
C00653=48.199,7.547,6.458,-177.7490,-19.5693,0.0000
C00654=48.453,5.301,6.447,-177.8170,-20.3344,0.0000
C00655=48.660,2.781,6.446,-178.7651,-20.4559,0.0000
C00656=48.740,0.000,6.447,179.9999,-20.4817,0.0000
C00657=48.660,-2.781,6.446,178.7652,-20.4559,0.0000
C00658=48.453,-5.301,6.447,177.8172,-20.3344,0.0000
C00659=48.199,-7.547,6.458,177.7489,-19.5692,0.0000
C00660=48.057,-9.067,6.484,179.0180,-17.5307,0.0000
C00661=48.028,-10.113,6.517,-179.6960,-14.2045,0.0000
C00662=48.058,-10.965,6.549,-179.4432,-10.3655,0.0000
C00663=48.078,-11.826,6.572,179.9179,-6.9386,0.0000
C00664=48.000,-12.898,6.582,179.4948,-4.0963,0.0000
C00665=47.771,-14.270,6.588,179.6240,-1.8276,0.0000
C00666=47.406,-15.768,6.592,179.8791,-0.4283,0.0000
C00667=46.944,-17.193,6.597,179.9722,-0.0771,0.0000
C00668=46.450,-18.501,6.600,179.9965,-0.0088,0.0000
C00669=45.928,-19.763,6.600,179.9962,-0.0087,0.0000
C00670=45.352,-21.037,6.597,179.9651,-0.0742,0.0000
C00671=44.670,-22.372,6.592,179.7826,-0.3883,0.0000
C00672=43.870,-23.689,6.588,178.9732,-1.5580,0.0000
C00673=43.061,-24.821,6.582,177.4573,-3.2521,0.0000
C00674=42.359,-25.634,6.572,175.1392,-4.9582,0.0000
C00675=41.735,-26.229,6.549,172.2431,-6.9191,0.0000
C00676=41.112,-26.810,6.517,169.6441,-9.7806,0.0000
C00677=40.393,-27.570,6.484,168.0701,-12.9763,0.0000
C00678=39.419,-28.746,6.458,167.3872,-15.2489,0.0000
C00679=38.009,-30.513,6.447,166.7599,-15.7223,0.0000
C00680=36.374,-32.441,6.446,166.0406,-15.1533,0.0000
C00681=34.464,-34.464,6.447,165.2049,-14.3250,0.0000
C00682=32.441,-36.374,6.446,164.4078,-13.4648,0.0000
C00683=30.513,-38.009,6.447,163.8706,-12.7364,0.0000
C00684=28.746,-39.419,6.458,164.3922,-12.1617,0.0000
C00685=27.570,-40.393,6.484,166.7472,-11.6210,0.0000
C00686=26.810,-41.112,6.517,170.0607,-10.2038,0.0000
C00687=26.229,-41.735,6.549,173.0177,-7.7000,0.0000
C00688=25.634,-42.359,6.572,175.0240,-4.8425,0.0000
C00689=24.821,-43.061,6.582,176.7447,-2.5386,0.0000
C00690=23.689,-43.870,6.588,178.4417,-1.0264,0.0000
C00691=22.372,-44.670,6.592,179.6117,-0.2174,0.0000
C00692=21.037,-45.352,6.597,179.9258,-0.0349,0.0000
C00693=19.763,-45.928,6.600,179.9913,-0.0038,0.0000
C00694=18.501,-46.450,6.600,179.9912,-0.0035,0.0000
C00695=17.193,-46.944,6.597,179.9229,-0.0278,0.0000
C00696=15.768,-47.406,6.592,179.5717,-0.1209,0.0000
C00697=14.270,-47.771,6.588,178.1724,-0.3758,0.0000
C00698=12.898,-48.000,6.582,175.9035,-0.5039,0.0000
C00699=11.826,-48.078,6.572,173.0614,-0.0815,0.0000
C00700=10.965,-48.058,6.549,169.6341,0.5477,0.0000
C00701=10.113,-48.028,6.517,165.7953,0.2947,0.0000
C00702=9.067,-48.057,6.484,162.4669,-0.9364,0.0000
C00703=7.547,-48.199,6.458,160.4168,-2.1209,0.0000
C00704=5.301,-48.453,6.447,159.6520,-2.0469,0.0000
C00705=2.781,-48.660,6.446,159.5397,-1.1571,0.0000
C00706=0.000,-48.740,6.447,159.5183,0.0001,0.0000
C00707=0.000,-48.740,6.447,159.5183,0.0001,0.0000
C00708=-2.781,-48.660,6.446,159.5397,1.1569,0.0000
C00709=-5.301,-48.453,6.447,159.6520,2.0467,0.0000
C00710=-7.547,-48.199,6.458,160.4168,2.1210,0.0000
C00711=-9.067,-48.057,6.484,162.4669,0.9364,0.0000
C00712=-10.113,-48.028,6.517,165.7953,-0.2947,0.0000
C00713=-10.965,-48.058,6.549,169.6341,-0.5477,0.0000
C00714=-11.826,-48.078,6.572,173.0614,0.0815,0.0000
C00715=-12.898,-48.000,6.582,175.9035,0.5039,0.0000
C00716=-14.270,-47.771,6.588,178.1724,0.3758,0.0000
C00717=-15.768,-47.406,6.592,179.5717,0.1209,0.0000
C00718=-17.193,-46.944,6.597,179.9229,0.0278,0.0000
C00719=-18.501,-46.450,6.600,179.9912,0.0035,0.0000
C00720=-19.763,-45.928,6.600,179.9913,0.0038,0.0000
C00721=-21.037,-45.352,6.597,179.9258,0.0349,0.0000
C00722=-22.372,-44.670,6.592,179.6117,0.2174,0.0000
C00723=-23.689,-43.870,6.588,178.4417,1.0264,0.0000
C00724=-24.821,-43.061,6.582,176.7447,2.5386,0.0000
C00725=-25.634,-42.359,6.572,175.0240,4.8425,0.0000
C00726=-26.229,-41.735,6.549,173.0177,7.7000,0.0000
C00727=-26.810,-41.112,6.517,170.0607,10.2038,0.0000
C00728=-27.570,-40.393,6.484,166.7472,11.6210,0.0000
C00729=-28.746,-39.419,6.458,164.3922,12.1618,0.0000
C00730=-30.513,-38.009,6.447,163.8705,12.7362,0.0000
C00731=-32.441,-36.374,6.446,164.4076,13.4647,0.0000
C00732=-34.464,-34.464,6.447,165.2050,14.3251,0.0000
C00733=-36.374,-32.441,6.446,166.0406,15.1532,0.0000
C00734=-38.009,-30.513,6.447,166.7598,15.7222,0.0000
C00735=-39.419,-28.746,6.458,167.3873,15.2489,0.0000
C00736=-40.393,-27.570,6.484,168.0701,12.9763,0.0000
C00737=-41.112,-26.810,6.517,169.6441,9.7806,0.0000
C00738=-41.735,-26.229,6.549,172.2431,6.9191,0.0000
C00739=-42.359,-25.634,6.572,175.1392,4.9582,0.0000
C00740=-43.061,-24.821,6.582,177.4573,3.2521,0.0000
C00741=-43.870,-23.689,6.588,178.9732,1.5580,0.0000
C00742=-44.670,-22.372,6.592,179.7826,0.3883,0.0000
C00743=-45.352,-21.037,6.597,179.9651,0.0742,0.0000
C00744=-45.928,-19.763,6.600,179.9962,0.0087,0.0000
C00745=-46.450,-18.501,6.600,179.9965,0.0088,0.0000
C00746=-46.944,-17.193,6.597,179.9722,0.0771,0.0000
C00747=-47.406,-15.768,6.592,179.8791,0.4283,0.0000
C00748=-47.771,-14.270,6.588,179.6240,1.8276,0.0000
C00749=-48.000,-12.898,6.582,179.4948,4.0963,0.0000
C00750=-48.078,-11.826,6.572,179.9179,6.9386,0.0000
C00751=-48.058,-10.965,6.549,-179.4432,10.3655,0.0000
C00752=-48.028,-10.113,6.517,-179.6960,14.2045,0.0000
C00753=-48.057,-9.067,6.484,179.0180,17.5307,0.0000
C00754=-48.199,-7.547,6.458,177.7490,19.5693,0.0000
C00755=-48.453,-5.301,6.447,177.8170,20.3344,0.0000
C00756=-48.660,-2.781,6.446,178.7651,20.4559,0.0000
C00757=-48.740,0.000,6.447,-179.9999,20.4817,0.0000
C00758=-48.660,2.781,6.446,-178.7652,20.4559,0.0000
C00759=-48.453,5.301,6.447,-177.8172,20.3344,0.0000
C00760=-48.199,7.547,6.458,-177.7489,19.5692,0.0000
C00761=-48.057,9.067,6.484,-179.0180,17.5307,0.0000
C00762=-48.028,10.113,6.517,179.6960,14.2045,0.0000
C00763=-48.058,10.965,6.549,179.4432,10.3655,0.0000
C00764=-48.078,11.826,6.572,-179.9179,6.9386,0.0000
C00765=-48.000,12.898,6.582,-179.4948,4.0963,0.0000
C00766=-47.771,14.270,6.588,-179.6240,1.8276,0.0000
C00767=-47.406,15.768,6.592,-179.8791,0.4283,0.0000
C00768=-46.944,17.193,6.597,-179.9722,0.0771,0.0000
C00769=-46.450,18.501,6.600,-179.9965,0.0088,0.0000
C00770=-45.928,19.763,6.600,-179.9962,0.0087,0.0000
C00771=-45.352,21.037,6.597,-179.9651,0.0742,0.0000
C00772=-44.670,22.372,6.592,-179.7826,0.3883,0.0000
C00773=-43.870,23.689,6.588,-178.9732,1.5580,0.0000
C00774=-43.061,24.821,6.582,-177.4573,3.2521,0.0000
C00775=-42.359,25.634,6.572,-175.1392,4.9582,0.0000
C00776=-41.735,26.229,6.549,-172.2431,6.9191,0.0000
C00777=-41.112,26.810,6.517,-169.6441,9.7806,0.0000
C00778=-40.393,27.570,6.484,-168.0701,12.9763,0.0000
C00779=-39.419,28.746,6.458,-167.3872,15.2489,0.0000
C00780=-38.009,30.513,6.447,-166.7599,15.7223,0.0000
C00781=-36.374,32.441,6.446,-166.0406,15.1533,0.0000
C00782=-34.464,34.464,6.447,-165.2049,14.3250,0.0000
C00783=-32.441,36.374,6.446,-164.4078,13.4648,0.0000
C00784=-30.513,38.009,6.447,-163.8706,12.7364,0.0000
C00785=-28.746,39.419,6.458,-164.3922,12.1617,0.0000
C00786=-27.570,40.393,6.484,-166.7472,11.6210,0.0000
C00787=-26.810,41.112,6.517,-170.0607,10.2038,0.0000
C00788=-26.229,41.735,6.549,-173.0177,7.7000,0.0000
C00789=-25.634,42.359,6.572,-175.0240,4.8425,0.0000
C00790=-24.821,43.061,6.582,-176.7447,2.5386,0.0000
C00791=-23.689,43.870,6.588,-178.4417,1.0264,0.0000
C00792=-22.372,44.670,6.592,-179.6117,0.2174,0.0000
C00793=-21.037,45.352,6.597,-179.9258,0.0349,0.0000
C00794=-19.763,45.928,6.600,-179.9913,0.0038,0.0000
C00795=-18.501,46.450,6.600,-179.9912,0.0035,0.0000
C00796=-17.193,46.944,6.597,-179.9229,0.0278,0.0000
C00797=-15.768,47.406,6.592,-179.5717,0.1209,0.0000
C00798=-14.270,47.771,6.588,-178.1724,0.3758,0.0000
C00799=-12.898,48.000,6.582,-175.9035,0.5039,0.0000
C00800=-11.826,48.078,6.572,-173.0614,0.0815,0.0000
C00801=-10.965,48.058,6.549,-169.6341,-0.5477,0.0000
C00802=-10.113,48.028,6.517,-165.7953,-0.2947,0.0000
C00803=-9.067,48.057,6.484,-162.4669,0.9364,0.0000
C00804=-7.547,48.199,6.458,-160.4168,2.1210,0.0000
C00805=-5.301,48.453,6.447,-159.6520,2.0467,0.0000
C00806=-2.781,48.660,6.446,-159.5397,1.1569,0.0000
C00807=0.000,48.740,6.447,-159.5183,0.0001,0.0000
C00808=0.000,47.885,8.473,-154.8794,0.0002,0.0000
C00809=2.703,47.807,8.473,-154.9046,-1.3964,0.0000
C00810=5.169,47.608,8.474,-155.0307,-2.3509,0.0000
C00811=7.387,47.387,8.496,-155.9336,-1.8012,0.0000
C00812=8.874,47.327,8.550,-158.8415,0.9445,0.0000
C00813=9.895,47.421,8.620,-163.9068,3.0310,0.0000
C00814=10.731,47.601,8.688,-169.0791,2.8184,0.0000
C00815=11.577,47.783,8.737,-172.7349,1.1937,0.0000
C00816=12.629,47.854,8.761,-175.6219,-0.0563,0.0000
C00817=14.018,47.741,8.773,-178.1277,-0.2591,0.0000
C00818=15.568,47.442,8.783,-179.6493,-0.0862,0.0000
C00819=17.067,46.986,8.793,-179.9232,-0.0272,0.0000
C00820=18.458,46.467,8.799,-179.9915,-0.0033,0.0000
C00821=19.805,45.909,8.799,-179.9916,-0.0037,0.0000
C00822=21.155,45.292,8.793,-179.9265,-0.0351,0.0000
C00823=22.539,44.555,8.783,-179.6910,-0.1870,0.0000
C00824=23.846,43.670,8.773,-178.4926,-1.1405,0.0000
C00825=24.908,42.767,8.761,-176.8614,-3.0544,0.0000
C00826=25.601,41.974,8.737,-175.6943,-5.9772,0.0000
C00827=26.071,41.247,8.688,-174.2337,-9.7047,0.0000
C00828=26.535,40.528,8.620,-170.6286,-13.4812,0.0000
C00829=27.190,39.740,8.550,-165.3625,-15.4769,0.0000
C00830=28.285,38.731,8.496,-161.2137,-15.4256,0.0000
C00831=30.009,37.319,8.474,-160.1357,-15.6188,0.0000
C00832=31.894,35.716,8.473,-160.6999,-16.4143,0.0000
C00833=33.859,33.859,8.473,-161.6576,-17.4688,0.0000
C00834=35.716,31.894,8.473,-162.6652,-18.4842,0.0000
C00835=37.319,30.009,8.474,-163.4455,-19.1015,0.0000
C00836=38.731,28.285,8.496,-163.7512,-18.0858,0.0000
C00837=39.740,27.190,8.550,-164.0300,-14.0955,0.0000
C00838=40.528,26.535,8.620,-166.3433,-9.1110,0.0000
C00839=41.247,26.071,8.688,-170.2468,-5.6835,0.0000
C00840=41.974,25.601,8.737,-174.0060,-4.2823,0.0000
C00841=42.767,24.908,8.761,-176.9411,-3.1341,0.0000
C00842=43.670,23.846,8.773,-178.8591,-1.5071,0.0000
C00843=44.555,22.539,8.783,-179.8130,-0.3090,0.0000
C00844=45.292,21.155,8.793,-179.9649,-0.0735,0.0000
C00845=45.909,19.805,8.799,-179.9963,-0.0084,0.0000
C00846=46.467,18.458,8.799,-179.9967,-0.0085,0.0000
C00847=46.986,17.067,8.793,-179.9728,-0.0768,0.0000
C00848=47.442,15.568,8.783,-179.9138,-0.3507,0.0000
C00849=47.741,14.018,8.773,-179.7407,-1.8723,0.0000
C00850=47.854,12.629,8.761,-179.9435,-4.3781,0.0000
C00851=47.783,11.577,8.737,178.7966,-7.2635,0.0000
C00852=47.601,10.731,8.688,177.1297,-10.9075,0.0000
C00853=47.421,9.895,8.620,176.8456,-16.0701,0.0000
C00854=47.327,8.874,8.550,178.9873,-21.1555,0.0000
C00855=47.387,7.387,8.496,-178.0274,-24.0538,0.0000
C00856=47.608,5.169,8.474,-177.4070,-24.9468,0.0000
C00857=47.807,2.703,8.473,-178.4581,-25.0874,0.0000
C00858=47.885,0.000,8.473,179.9998,-25.1206,0.0000
C00859=47.807,-2.703,8.473,178.4583,-25.0874,0.0000
C00860=47.608,-5.169,8.474,177.4073,-24.9468,0.0000
C00861=47.387,-7.387,8.496,178.0272,-24.0537,0.0000
C00862=47.327,-8.874,8.550,-178.9873,-21.1555,0.0000
C00863=47.421,-9.895,8.620,-176.8456,-16.0701,0.0000
C00864=47.601,-10.731,8.688,-177.1297,-10.9075,0.0000
C00865=47.783,-11.577,8.737,-178.7966,-7.2635,0.0000
C00866=47.854,-12.629,8.761,179.9435,-4.3781,0.0000
C00867=47.741,-14.018,8.773,179.7407,-1.8723,0.0000
C00868=47.442,-15.568,8.783,179.9138,-0.3507,0.0000
C00869=46.986,-17.067,8.793,179.9728,-0.0768,0.0000
C00870=46.467,-18.458,8.799,179.9967,-0.0085,0.0000
C00871=45.909,-19.805,8.799,179.9963,-0.0084,0.0000
C00872=45.292,-21.155,8.793,179.9649,-0.0735,0.0000
C00873=44.555,-22.539,8.783,179.8130,-0.3090,0.0000
C00874=43.670,-23.846,8.773,178.8591,-1.5071,0.0000
C00875=42.767,-24.908,8.761,176.9411,-3.1341,0.0000
C00876=41.974,-25.601,8.737,174.0060,-4.2823,0.0000
C00877=41.247,-26.071,8.688,170.2468,-5.6835,0.0000
C00878=40.528,-26.535,8.620,166.3433,-9.1110,0.0000
C00879=39.740,-27.190,8.550,164.0300,-14.0955,0.0000
C00880=38.731,-28.285,8.496,163.7510,-18.0857,0.0000
C00881=37.319,-30.009,8.474,163.4457,-19.1017,0.0000
C00882=35.716,-31.894,8.473,162.6653,-18.4844,0.0000
C00883=33.859,-33.859,8.473,161.6573,-17.4685,0.0000
C00884=31.894,-35.716,8.473,160.7001,-16.4145,0.0000
C00885=30.009,-37.319,8.474,160.1359,-15.6190,0.0000
C00886=28.285,-38.731,8.496,161.2136,-15.4254,0.0000
C00887=27.190,-39.740,8.550,165.3625,-15.4769,0.0000
C00888=26.535,-40.528,8.620,170.6286,-13.4812,0.0000
C00889=26.071,-41.247,8.688,174.2337,-9.7047,0.0000
C00890=25.601,-41.974,8.737,175.6943,-5.9772,0.0000
C00891=24.908,-42.767,8.761,176.8614,-3.0544,0.0000
C00892=23.846,-43.670,8.773,178.4926,-1.1405,0.0000
C00893=22.539,-44.555,8.783,179.6910,-0.1870,0.0000
C00894=21.155,-45.292,8.793,179.9265,-0.0351,0.0000
C00895=19.805,-45.909,8.799,179.9916,-0.0037,0.0000
C00896=18.458,-46.467,8.799,179.9915,-0.0033,0.0000
C00897=17.067,-46.986,8.793,179.9232,-0.0272,0.0000
C00898=15.568,-47.442,8.783,179.6493,-0.0862,0.0000
C00899=14.018,-47.741,8.773,178.1277,-0.2591,0.0000
C00900=12.629,-47.854,8.761,175.6219,-0.0563,0.0000
C00901=11.577,-47.783,8.737,172.7349,1.1937,0.0000
C00902=10.731,-47.601,8.688,169.0791,2.8184,0.0000
C00903=9.895,-47.421,8.620,163.9068,3.0310,0.0000
C00904=8.874,-47.327,8.550,158.8415,0.9445,0.0000
C00905=7.387,-47.387,8.496,155.9336,-1.8012,0.0000
C00906=5.169,-47.608,8.474,155.0307,-2.3509,0.0000
C00907=2.703,-47.807,8.473,154.9046,-1.3964,0.0000
C00908=0.000,-47.885,8.473,154.8794,0.0002,0.0000
C00909=0.000,-47.885,8.473,154.8794,0.0002,0.0000
C00910=-2.703,-47.807,8.473,154.9046,1.3962,0.0000
C00911=-5.169,-47.608,8.474,155.0307,2.3506,0.0000
C00912=-7.387,-47.387,8.496,155.9336,1.8014,0.0000
C00913=-8.874,-47.327,8.550,158.8415,-0.9445,0.0000
C00914=-9.895,-47.421,8.620,163.9068,-3.0310,0.0000
C00915=-10.731,-47.601,8.688,169.0791,-2.8184,0.0000
C00916=-11.577,-47.783,8.737,172.7349,-1.1937,0.0000
C00917=-12.629,-47.854,8.761,175.6219,0.0563,0.0000
C00918=-14.018,-47.741,8.773,178.1277,0.2591,0.0000
C00919=-15.568,-47.442,8.783,179.6493,0.0862,0.0000
C00920=-17.067,-46.986,8.793,179.9232,0.0272,0.0000
C00921=-18.458,-46.467,8.799,179.9915,0.0033,0.0000
C00922=-19.805,-45.909,8.799,179.9916,0.0037,0.0000
C00923=-21.155,-45.292,8.793,179.9265,0.0351,0.0000
C00924=-22.539,-44.555,8.783,179.6910,0.1870,0.0000
C00925=-23.846,-43.670,8.773,178.4926,1.1405,0.0000
C00926=-24.908,-42.767,8.761,176.8614,3.0544,0.0000
C00927=-25.601,-41.974,8.737,175.6943,5.9772,0.0000
C00928=-26.071,-41.247,8.688,174.2337,9.7047,0.0000
C00929=-26.535,-40.528,8.620,170.6286,13.4812,0.0000
C00930=-27.190,-39.740,8.550,165.3625,15.4769,0.0000
C00931=-28.285,-38.731,8.496,161.2137,15.4256,0.0000
C00932=-30.009,-37.319,8.474,160.1357,15.6188,0.0000
C00933=-31.894,-35.716,8.473,160.6999,16.4143,0.0000
C00934=-33.859,-33.859,8.473,161.6576,17.4688,0.0000
C00935=-35.716,-31.894,8.473,162.6652,18.4842,0.0000
C00936=-37.319,-30.009,8.474,163.4455,19.1015,0.0000
C00937=-38.731,-28.285,8.496,163.7512,18.0858,0.0000
C00938=-39.740,-27.190,8.550,164.0300,14.0955,0.0000
C00939=-40.528,-26.535,8.620,166.3433,9.1110,0.0000
C00940=-41.247,-26.071,8.688,170.2468,5.6835,0.0000
C00941=-41.974,-25.601,8.737,174.0060,4.2823,0.0000
C00942=-42.767,-24.908,8.761,176.9411,3.1341,0.0000
C00943=-43.670,-23.846,8.773,178.8591,1.5071,0.0000
C00944=-44.555,-22.539,8.783,179.8130,0.3090,0.0000
C00945=-45.292,-21.155,8.793,179.9649,0.0735,0.0000
C00946=-45.909,-19.805,8.799,179.9963,0.0084,0.0000
C00947=-46.467,-18.458,8.799,179.9967,0.0085,0.0000
C00948=-46.986,-17.067,8.793,179.9728,0.0768,0.0000
C00949=-47.442,-15.568,8.783,179.9138,0.3507,0.0000
C00950=-47.741,-14.018,8.773,179.7407,1.8723,0.0000
C00951=-47.854,-12.629,8.761,179.9435,4.3781,0.0000
C00952=-47.783,-11.577,8.737,-178.7966,7.2635,0.0000
C00953=-47.601,-10.731,8.688,-177.1297,10.9075,0.0000
C00954=-47.421,-9.895,8.620,-176.8456,16.0701,0.0000
C00955=-47.327,-8.874,8.550,-178.9873,21.1555,0.0000
C00956=-47.387,-7.387,8.496,178.0274,24.0538,0.0000
C00957=-47.608,-5.169,8.474,177.4070,24.9468,0.0000
C00958=-47.807,-2.703,8.473,178.4581,25.0874,0.0000
C00959=-47.885,0.000,8.473,-179.9998,25.1206,0.0000
C00960=-47.807,2.703,8.473,-178.4583,25.0874,0.0000
C00961=-47.608,5.169,8.474,-177.4073,24.9468,0.0000
C00962=-47.387,7.387,8.496,-178.0272,24.0537,0.0000
C00963=-47.327,8.874,8.550,178.9873,21.1555,0.0000
C00964=-47.421,9.895,8.620,176.8456,16.0701,0.0000
C00965=-47.601,10.731,8.688,177.1297,10.9075,0.0000
C00966=-47.783,11.577,8.737,178.7966,7.2635,0.0000
C00967=-47.854,12.629,8.761,-179.9435,4.3781,0.0000
C00968=-47.741,14.018,8.773,-179.7407,1.8723,0.0000
C00969=-47.442,15.568,8.783,-179.9138,0.3507,0.0000
C00970=-46.986,17.067,8.793,-179.9728,0.0768,0.0000
C00971=-46.467,18.458,8.799,-179.9967,0.0085,0.0000
C00972=-45.909,19.805,8.799,-179.9963,0.0084,0.0000
C00973=-45.292,21.155,8.793,-179.9649,0.0735,0.0000
C00974=-44.555,22.539,8.783,-179.8130,0.3090,0.0000
C00975=-43.670,23.846,8.773,-178.8591,1.5071,0.0000
C00976=-42.767,24.908,8.761,-176.9411,3.1341,0.0000
C00977=-41.974,25.601,8.737,-174.0060,4.2823,0.0000
C00978=-41.247,26.071,8.688,-170.2468,5.6835,0.0000
C00979=-40.528,26.535,8.620,-166.3433,9.1110,0.0000
C00980=-39.740,27.190,8.550,-164.0300,14.0955,0.0000
C00981=-38.731,28.285,8.496,-163.7510,18.0857,0.0000
C00982=-37.319,30.009,8.474,-163.4457,19.1017,0.0000
C00983=-35.716,31.894,8.473,-162.6653,18.4844,0.0000
C00984=-33.859,33.859,8.473,-161.6573,17.4685,0.0000
C00985=-31.894,35.716,8.473,-160.7001,16.4145,0.0000
C00986=-30.009,37.319,8.474,-160.1359,15.6190,0.0000
C00987=-28.285,38.731,8.496,-161.2136,15.4254,0.0000
C00988=-27.190,39.740,8.550,-165.3625,15.4769,0.0000
C00989=-26.535,40.528,8.620,-170.6286,13.4812,0.0000
C00990=-26.071,41.247,8.688,-174.2337,9.7047,0.0000
C00991=-25.601,41.974,8.737,-175.6943,5.9772,0.0000
C00992=-24.908,42.767,8.761,-176.8614,3.0544,0.0000
C00993=-23.846,43.670,8.773,-178.4926,1.1405,0.0000
C00994=-22.539,44.555,8.783,-179.6910,0.1870,0.0000
C00995=-21.155,45.292,8.793,-179.9265,0.0351,0.0000
C00996=-19.805,45.909,8.799,-179.9916,0.0037,0.0000
C00997=-18.458,46.467,8.799,-179.9915,0.0033,0.0000
C00998=-17.067,46.986,8.793,-179.9232,0.0272,0.0000
C00999=-15.568,47.442,8.783,-179.6493,0.0862,0.0000
C01000=-14.018,47.741,8.773,-178.1277,0.2591,0.0000
C01001=-12.629,47.854,8.761,-175.6219,0.0563,0.0000
C01002=-11.577,47.783,8.737,-172.7349,-1.1937,0.0000
C01003=-10.731,47.601,8.688,-169.0791,-2.8184,0.0000
C01004=-9.895,47.421,8.620,-163.9068,-3.0310,0.0000
C01005=-8.874,47.327,8.550,-158.8415,-0.9445,0.0000
C01006=-7.387,47.387,8.496,-155.9336,1.8014,0.0000
C01007=-5.169,47.608,8.474,-155.0307,2.3506,0.0000
C01008=-2.703,47.807,8.473,-154.9046,1.3962,0.0000
C01009=0.000,47.885,8.473,-154.8794,0.0002,0.0000
C01010=0.000,46.884,10.433,-151.1653,0.0002,0.0000
C01011=2.611,46.810,10.432,-151.1930,-1.5762,0.0000
C01012=5.015,46.620,10.433,-151.3262,-2.4871,0.0000
C01013=7.199,46.436,10.471,-152.3977,-0.9762,0.0000
C01014=8.646,46.466,10.562,-156.8195,3.8339,0.0000
C01015=9.635,46.699,10.682,-164.4281,6.1357,0.0000
C01016=10.451,47.054,10.800,-170.7349,4.7296,0.0000
C01017=11.278,47.426,10.887,-173.9779,2.3147,0.0000
C01018=12.303,47.677,10.929,-176.1454,0.4711,0.0000
C01019=13.711,47.704,10.951,-178.4247,-0.0968,0.0000
C01020=15.325,47.486,10.969,-179.8437,-0.0322,0.0000
C01021=16.914,47.036,10.987,-179.9356,-0.0223,0.0000
C01022=18.406,46.487,10.998,-179.9932,-0.0027,0.0000
C01023=19.856,45.886,10.998,-179.9933,-0.0029,0.0000
C01024=21.300,45.220,10.987,-179.9387,-0.0298,0.0000
C01025=22.741,44.414,10.969,-179.8667,-0.0878,0.0000
C01026=24.036,43.427,10.951,-178.8175,-1.0454,0.0000
C01027=25.013,42.412,10.929,-177.6055,-3.0580,0.0000
C01028=25.561,41.510,10.887,-177.3745,-5.8937,0.0000
C01029=25.882,40.662,10.800,-176.7905,-9.8902,0.0000
C01030=26.208,39.834,10.682,-173.2620,-15.3261,0.0000
C01031=26.743,38.970,10.562,-165.8972,-18.9653,0.0000
C01032=27.744,37.925,10.471,-159.0282,-18.3929,0.0000
C01033=29.419,36.512,10.433,-157.1341,-17.9557,0.0000
C01034=31.253,34.946,10.432,-157.6547,-18.7324,0.0000
C01035=33.152,33.152,10.433,-158.7295,-19.9396,0.0000
C01036=34.946,31.253,10.432,-159.8646,-21.1029,0.0000
C01037=36.512,29.419,10.433,-160.6227,-21.6937,0.0000
C01038=37.925,27.744,10.471,-160.3991,-19.8542,0.0000
C01039=38.970,26.743,10.562,-160.4893,-13.3227,0.0000
C01040=39.834,26.208,10.682,-164.5724,-6.4973,0.0000
C01041=40.662,25.882,10.800,-170.0945,-3.1618,0.0000
C01042=41.510,25.561,10.887,-174.1002,-2.6116,0.0000
C01043=42.412,25.013,10.929,-176.9394,-2.3911,0.0000
C01044=43.427,24.036,10.951,-178.9544,-1.1823,0.0000
C01045=44.414,22.741,10.969,-179.9122,-0.1333,0.0000
C01046=45.220,21.300,10.987,-179.9702,-0.0613,0.0000
C01047=45.886,19.856,10.998,-179.9971,-0.0067,0.0000
C01048=46.487,18.406,10.998,-179.9973,-0.0068,0.0000
C01049=47.036,16.914,10.987,-179.9777,-0.0644,0.0000
C01050=47.486,15.325,10.969,-179.9678,-0.1563,0.0000
C01051=47.704,13.711,10.951,-179.9032,-1.5753,0.0000
C01052=47.677,12.303,10.929,179.5279,-3.8544,0.0000
C01053=47.426,11.278,10.887,177.6724,-6.0172,0.0000
C01054=47.054,10.451,10.800,175.2082,-9.2332,0.0000
C01055=46.699,9.635,10.682,173.6324,-15.4805,0.0000
C01056=46.466,8.646,10.562,175.8305,-23.1256,0.0000
C01057=46.436,7.199,10.471,-178.8985,-27.5980,0.0000
C01058=46.620,5.015,10.433,-177.1658,-28.6443,0.0000
C01059=46.810,2.611,10.432,-178.2014,-28.7951,0.0000
C01060=46.884,0.000,10.433,179.9997,-28.8347,0.0000
C01061=46.810,-2.611,10.432,178.2017,-28.7951,0.0000
C01062=46.620,-5.015,10.433,177.1664,-28.6443,0.0000
C01063=46.436,-7.199,10.471,178.8981,-27.5980,0.0000
C01064=46.466,-8.646,10.562,-175.8305,-23.1256,0.0000
C01065=46.699,-9.635,10.682,-173.6324,-15.4805,0.0000
C01066=47.054,-10.451,10.800,-175.2082,-9.2332,0.0000
C01067=47.426,-11.278,10.887,-177.6724,-6.0172,0.0000
C01068=47.677,-12.303,10.929,-179.5279,-3.8544,0.0000
C01069=47.704,-13.711,10.951,179.9032,-1.5753,0.0000
C01070=47.486,-15.325,10.969,179.9678,-0.1563,0.0000
C01071=47.036,-16.914,10.987,179.9777,-0.0644,0.0000
C01072=46.487,-18.406,10.998,179.9973,-0.0068,0.0000
C01073=45.886,-19.856,10.998,179.9971,-0.0067,0.0000
C01074=45.220,-21.300,10.987,179.9702,-0.0613,0.0000
C01075=44.414,-22.741,10.969,179.9122,-0.1333,0.0000
C01076=43.427,-24.036,10.951,178.9544,-1.1823,0.0000
C01077=42.412,-25.013,10.929,176.9394,-2.3911,0.0000
C01078=41.510,-25.561,10.887,174.1002,-2.6116,0.0000
C01079=40.662,-25.882,10.800,170.0945,-3.1618,0.0000
C01080=39.834,-26.208,10.682,164.5724,-6.4973,0.0000
C01081=38.970,-26.743,10.562,160.4893,-13.3227,0.0000
C01082=37.925,-27.744,10.471,160.3988,-19.8540,0.0000
C01083=36.512,-29.419,10.433,160.6231,-21.6940,0.0000
C01084=34.946,-31.253,10.432,159.8649,-21.1031,0.0000
C01085=33.152,-33.152,10.433,158.7292,-19.9393,0.0000
C01086=31.253,-34.946,10.432,157.6550,-18.7327,0.0000
C01087=29.419,-36.512,10.433,157.1345,-17.9561,0.0000
C01088=27.744,-37.925,10.471,159.0280,-18.3926,0.0000
C01089=26.743,-38.970,10.562,165.8972,-18.9653,0.0000
C01090=26.208,-39.834,10.682,173.2620,-15.3261,0.0000
C01091=25.882,-40.662,10.800,176.7905,-9.8902,0.0000
C01092=25.561,-41.510,10.887,177.3745,-5.8937,0.0000
C01093=25.013,-42.412,10.929,177.6055,-3.0580,0.0000
C01094=24.036,-43.427,10.951,178.8175,-1.0454,0.0000
C01095=22.741,-44.414,10.969,179.8667,-0.0878,0.0000
C01096=21.300,-45.220,10.987,179.9387,-0.0298,0.0000
C01097=19.856,-45.886,10.998,179.9933,-0.0029,0.0000
C01098=18.406,-46.487,10.998,179.9932,-0.0027,0.0000
C01099=16.914,-47.036,10.987,179.9356,-0.0223,0.0000
C01100=15.325,-47.486,10.969,179.8437,-0.0322,0.0000
C01101=13.711,-47.704,10.951,178.4247,-0.0968,0.0000
C01102=12.303,-47.677,10.929,176.1454,0.4711,0.0000
C01103=11.278,-47.426,10.887,173.9779,2.3147,0.0000
C01104=10.451,-47.054,10.800,170.7349,4.7296,0.0000
C01105=9.635,-46.699,10.682,164.4281,6.1357,0.0000
C01106=8.646,-46.466,10.562,156.8195,3.8339,0.0000
C01107=7.199,-46.436,10.471,152.3977,-0.9762,0.0000
C01108=5.015,-46.620,10.433,151.3262,-2.4871,0.0000
C01109=2.611,-46.810,10.432,151.1930,-1.5762,0.0000
C01110=0.000,-46.884,10.433,151.1653,0.0002,0.0000
C01111=0.000,-46.884,10.433,151.1653,0.0002,0.0000
C01112=-2.611,-46.810,10.432,151.1930,1.5758,0.0000
C01113=-5.015,-46.620,10.433,151.3262,2.4866,0.0000
C01114=-7.199,-46.436,10.471,152.3977,0.9765,0.0000
C01115=-8.646,-46.466,10.562,156.8195,-3.8339,0.0000
C01116=-9.635,-46.699,10.682,164.4281,-6.1357,0.0000
C01117=-10.451,-47.054,10.800,170.7349,-4.7296,0.0000
C01118=-11.278,-47.426,10.887,173.9779,-2.3147,0.0000
C01119=-12.303,-47.677,10.929,176.1454,-0.4711,0.0000
C01120=-13.711,-47.704,10.951,178.4247,0.0968,0.0000
C01121=-15.325,-47.486,10.969,179.8437,0.0322,0.0000
C01122=-16.914,-47.036,10.987,179.9356,0.0223,0.0000
C01123=-18.406,-46.487,10.998,179.9932,0.0027,0.0000
C01124=-19.856,-45.886,10.998,179.9933,0.0029,0.0000
C01125=-21.300,-45.220,10.987,179.9387,0.0298,0.0000
C01126=-22.741,-44.414,10.969,179.8667,0.0878,0.0000
C01127=-24.036,-43.427,10.951,178.8175,1.0454,0.0000
C01128=-25.013,-42.412,10.929,177.6055,3.0580,0.0000
C01129=-25.561,-41.510,10.887,177.3745,5.8937,0.0000
C01130=-25.882,-40.662,10.800,176.7905,9.8902,0.0000
C01131=-26.208,-39.834,10.682,173.2620,15.3261,0.0000
C01132=-26.743,-38.970,10.562,165.8972,18.9653,0.0000
C01133=-27.744,-37.925,10.471,159.0282,18.3929,0.0000
C01134=-29.419,-36.512,10.433,157.1341,17.9557,0.0000
C01135=-31.253,-34.946,10.432,157.6547,18.7324,0.0000
C01136=-33.152,-33.152,10.433,158.7295,19.9396,0.0000
C01137=-34.946,-31.253,10.432,159.8646,21.1029,0.0000
C01138=-36.512,-29.419,10.433,160.6227,21.6937,0.0000
C01139=-37.925,-27.744,10.471,160.3991,19.8542,0.0000
C01140=-38.970,-26.743,10.562,160.4893,13.3227,0.0000
C01141=-39.834,-26.208,10.682,164.5724,6.4973,0.0000
C01142=-40.662,-25.882,10.800,170.0945,3.1618,0.0000
C01143=-41.510,-25.561,10.887,174.1002,2.6116,0.0000
C01144=-42.412,-25.013,10.929,176.9394,2.3911,0.0000
C01145=-43.427,-24.036,10.951,178.9544,1.1823,0.0000
C01146=-44.414,-22.741,10.969,179.9122,0.1333,0.0000
C01147=-45.220,-21.300,10.987,179.9702,0.0613,0.0000
C01148=-45.886,-19.856,10.998,179.9971,0.0067,0.0000
C01149=-46.487,-18.406,10.998,179.9973,0.0068,0.0000
C01150=-47.036,-16.914,10.987,179.9777,0.0644,0.0000
C01151=-47.486,-15.325,10.969,179.9678,0.1563,0.0000
C01152=-47.704,-13.711,10.951,179.9032,1.5753,0.0000
C01153=-47.677,-12.303,10.929,-179.5279,3.8544,0.0000
C01154=-47.426,-11.278,10.887,-177.6724,6.0172,0.0000
C01155=-47.054,-10.451,10.800,-175.2082,9.2332,0.0000
C01156=-46.699,-9.635,10.682,-173.6324,15.4805,0.0000
C01157=-46.466,-8.646,10.562,-175.8305,23.1256,0.0000
C01158=-46.436,-7.199,10.471,178.8985,27.5980,0.0000
C01159=-46.620,-5.015,10.433,177.1658,28.6443,0.0000
C01160=-46.810,-2.611,10.432,178.2014,28.7951,0.0000
C01161=-46.884,0.000,10.433,-179.9997,28.8347,0.0000
C01162=-46.810,2.611,10.432,-178.2017,28.7951,0.0000
C01163=-46.620,5.015,10.433,-177.1664,28.6443,0.0000
C01164=-46.436,7.199,10.471,-178.8981,27.5980,0.0000
C01165=-46.466,8.646,10.562,175.8305,23.1256,0.0000
C01166=-46.699,9.635,10.682,173.6324,15.4805,0.0000
C01167=-47.054,10.451,10.800,175.2082,9.2332,0.0000
C01168=-47.426,11.278,10.887,177.6724,6.0172,0.0000
C01169=-47.677,12.303,10.929,179.5279,3.8544,0.0000
C01170=-47.704,13.711,10.951,-179.9032,1.5753,0.0000
C01171=-47.486,15.325,10.969,-179.9678,0.1563,0.0000
C01172=-47.036,16.914,10.987,-179.9777,0.0644,0.0000
C01173=-46.487,18.406,10.998,-179.9973,0.0068,0.0000
C01174=-45.886,19.856,10.998,-179.9971,0.0067,0.0000
C01175=-45.220,21.300,10.987,-179.9702,0.0613,0.0000
C01176=-44.414,22.741,10.969,-179.9122,0.1333,0.0000
C01177=-43.427,24.036,10.951,-178.9544,1.1823,0.0000
C01178=-42.412,25.013,10.929,-176.9394,2.3911,0.0000
C01179=-41.510,25.561,10.887,-174.1002,2.6116,0.0000
C01180=-40.662,25.882,10.800,-170.0945,3.1618,0.0000
C01181=-39.834,26.208,10.682,-164.5724,6.4973,0.0000
C01182=-38.970,26.743,10.562,-160.4893,13.3227,0.0000
C01183=-37.925,27.744,10.471,-160.3988,19.8540,0.0000
C01184=-36.512,29.419,10.433,-160.6231,21.6940,0.0000
C01185=-34.946,31.253,10.432,-159.8649,21.1031,0.0000
C01186=-33.152,33.152,10.433,-158.7292,19.9393,0.0000
C01187=-31.253,34.946,10.432,-157.6550,18.7327,0.0000
C01188=-29.419,36.512,10.433,-157.1345,17.9561,0.0000
C01189=-27.744,37.925,10.471,-159.0280,18.3926,0.0000
C01190=-26.743,38.970,10.562,-165.8972,18.9653,0.0000
C01191=-26.208,39.834,10.682,-173.2620,15.3261,0.0000
C01192=-25.882,40.662,10.800,-176.7905,9.8902,0.0000
C01193=-25.561,41.510,10.887,-177.3745,5.8937,0.0000
C01194=-25.013,42.412,10.929,-177.6055,3.0580,0.0000
C01195=-24.036,43.427,10.951,-178.8175,1.0454,0.0000
C01196=-22.741,44.414,10.969,-179.8667,0.0878,0.0000
C01197=-21.300,45.220,10.987,-179.9387,0.0298,0.0000
C01198=-19.856,45.886,10.998,-179.9933,0.0029,0.0000
C01199=-18.406,46.487,10.998,-179.9932,0.0027,0.0000
C01200=-16.914,47.036,10.987,-179.9356,0.0223,0.0000
C01201=-15.325,47.486,10.969,-179.8437,0.0322,0.0000
C01202=-13.711,47.704,10.951,-178.4247,0.0968,0.0000
C01203=-12.303,47.677,10.929,-176.1454,-0.4711,0.0000
C01204=-11.278,47.426,10.887,-173.9779,-2.3147,0.0000
C01205=-10.451,47.054,10.800,-170.7349,-4.7296,0.0000
C01206=-9.635,46.699,10.682,-164.4281,-6.1357,0.0000
C01207=-8.646,46.466,10.562,-156.8195,-3.8339,0.0000
C01208=-7.199,46.436,10.471,-152.3977,0.9765,0.0000
C01209=-5.015,46.620,10.433,-151.3262,2.4866,0.0000
C01210=-2.611,46.810,10.432,-151.1930,1.5758,0.0000
C01211=0.000,46.884,10.433,-151.1653,0.0002,0.0000
C01212=0.000,45.772,12.331,-148.2173,0.0003,0.0000
C01213=2.510,45.702,12.329,-148.2466,-1.7081,0.0000
C01214=4.844,45.521,12.332,-148.3842,-2.4822,0.0000
C01215=6.990,45.375,12.387,-149.7196,0.2799,0.0000
C01216=8.390,45.503,12.523,-156.6479,7.2043,0.0000
C01217=9.343,45.885,12.705,-167.0222,8.2576,0.0000
C01218=10.132,46.432,12.887,-173.6461,5.1271,0.0000
C01219=10.935,47.018,13.022,-176.2893,2.4011,0.0000
C01220=11.930,47.474,13.088,-177.4312,0.7183,0.0000
C01221=13.360,47.661,13.123,-179.0290,0.0208,0.0000
C01222=15.047,47.537,13.151,179.8657,0.0220,0.0000
C01223=16.738,47.094,13.179,-179.9573,-0.0145,0.0000
C01224=18.347,46.510,13.197,-179.9960,-0.0016,0.0000
C01225=19.915,45.860,13.197,-179.9960,-0.0018,0.0000
C01226=21.465,45.136,13.179,-179.9596,-0.0199,0.0000
C01227=22.974,44.253,13.151,179.8895,0.0794,0.0000
C01228=24.255,43.149,13.123,-179.3281,-0.7013,0.0000
C01229=25.133,42.005,13.088,-178.6911,-2.3242,0.0000
C01230=25.514,40.979,13.022,-179.0750,-4.3212,0.0000
C01231=25.668,39.997,12.887,-179.1463,-8.1134,0.0000
C01232=25.839,39.052,12.705,-176.7006,-14.9934,0.0000
C01233=26.243,38.108,12.523,-168.2536,-21.5152,0.0000
C01234=27.143,37.028,12.387,-157.7615,-21.0999,0.0000
C01235=28.763,35.614,12.332,-154.7665,-19.8591,0.0000
C01236=30.541,34.091,12.329,-155.1829,-20.5413,0.0000
C01237=32.366,32.366,12.331,-156.3406,-21.8659,0.0000
C01238=34.091,30.541,12.329,-157.5673,-23.1433,0.0000
C01239=35.614,28.763,12.332,-158.2333,-23.6374,0.0000
C01240=37.028,27.143,12.387,-157.3703,-20.6767,0.0000
C01241=38.108,26.243,12.523,-158.0679,-10.9174,0.0000
C01242=39.052,25.839,12.705,-164.9828,-3.1869,0.0000
C01243=39.997,25.668,12.887,-171.8857,-0.8452,0.0000
C01244=40.979,25.514,13.022,-175.6783,-0.9224,0.0000
C01245=42.005,25.133,13.088,-177.6752,-1.3079,0.0000
C01246=43.149,24.255,13.123,-179.2987,-0.6719,0.0000
C01247=44.253,22.974,13.151,179.9206,0.1105,0.0000
C01248=45.136,21.465,13.179,-179.9801,-0.0404,0.0000
C01249=45.860,19.915,13.197,-179.9982,-0.0040,0.0000
C01250=46.510,18.347,13.197,-179.9984,-0.0040,0.0000
C01251=47.094,16.738,13.179,-179.9855,-0.0427,0.0000
C01252=47.537,15.047,13.151,179.9780,0.1343,0.0000
C01253=47.661,13.360,13.123,179.9792,-0.9710,0.0000
C01254=47.474,11.930,13.088,179.2810,-2.5686,0.0000
C01255=47.018,10.935,13.022,177.5938,-3.7074,0.0000
C01256=46.432,10.132,12.887,174.8414,-6.3283,0.0000
C01257=45.885,9.343,12.705,171.5291,-12.8409,0.0000
C01258=45.503,8.390,12.523,172.1606,-23.1570,0.0000
C01259=45.375,6.990,12.387,179.6759,-30.2800,0.0000
C01260=45.521,4.844,12.332,-177.0859,-31.5827,0.0000
C01261=45.702,2.510,12.329,-177.9915,-31.7377,0.0000
C01262=45.772,0.000,12.331,179.9996,-31.7827,0.0000
C01263=45.702,-2.510,12.329,177.9919,-31.7377,0.0000
C01264=45.521,-4.844,12.332,177.0867,-31.5827,0.0000
C01265=45.375,-6.990,12.387,-179.6765,-30.2800,0.0000
C01266=45.503,-8.390,12.523,-172.1606,-23.1570,0.0000
C01267=45.885,-9.343,12.705,-171.5291,-12.8409,0.0000
C01268=46.432,-10.132,12.887,-174.8414,-6.3283,0.0000
C01269=47.018,-10.935,13.022,-177.5938,-3.7074,0.0000
C01270=47.474,-11.930,13.088,-179.2810,-2.5686,0.0000
C01271=47.661,-13.360,13.123,-179.9792,-0.9710,0.0000
C01272=47.537,-15.047,13.151,-179.9780,0.1343,0.0000
C01273=47.094,-16.738,13.179,179.9855,-0.0427,0.0000
C01274=46.510,-18.347,13.197,179.9984,-0.0040,0.0000
C01275=45.860,-19.915,13.197,179.9982,-0.0040,0.0000
C01276=45.136,-21.465,13.179,179.9801,-0.0404,0.0000
C01277=44.253,-22.974,13.151,-179.9206,0.1105,0.0000
C01278=43.149,-24.255,13.123,179.2987,-0.6719,0.0000
C01279=42.005,-25.133,13.088,177.6752,-1.3079,0.0000
C01280=40.979,-25.514,13.022,175.6783,-0.9224,0.0000
C01281=39.997,-25.668,12.887,171.8857,-0.8452,0.0000
C01282=39.052,-25.839,12.705,164.9828,-3.1869,0.0000
C01283=38.108,-26.243,12.523,158.0679,-10.9174,0.0000
C01284=37.028,-27.143,12.387,157.3700,-20.6763,0.0000
C01285=35.614,-28.763,12.332,158.2337,-23.6380,0.0000
C01286=34.091,-30.541,12.329,157.5676,-23.1436,0.0000
C01287=32.366,-32.366,12.331,156.3402,-21.8655,0.0000
C01288=30.541,-34.091,12.329,155.1831,-20.5417,0.0000
C01289=28.763,-35.614,12.332,154.7670,-19.8596,0.0000
C01290=27.143,-37.028,12.387,157.7612,-21.0996,0.0000
C01291=26.243,-38.108,12.523,168.2536,-21.5152,0.0000
C01292=25.839,-39.052,12.705,176.7006,-14.9934,0.0000
C01293=25.668,-39.997,12.887,179.1463,-8.1134,0.0000
C01294=25.514,-40.979,13.022,179.0750,-4.3212,0.0000
C01295=25.133,-42.005,13.088,178.6911,-2.3242,0.0000
C01296=24.255,-43.149,13.123,179.3281,-0.7013,0.0000
C01297=22.974,-44.253,13.151,-179.8895,0.0794,0.0000
C01298=21.465,-45.136,13.179,179.9596,-0.0199,0.0000
C01299=19.915,-45.860,13.197,179.9960,-0.0018,0.0000
C01300=18.347,-46.510,13.197,179.9960,-0.0016,0.0000
C01301=16.738,-47.094,13.179,179.9573,-0.0145,0.0000
C01302=15.047,-47.537,13.151,-179.8657,0.0220,0.0000
C01303=13.360,-47.661,13.123,179.0290,0.0208,0.0000
C01304=11.930,-47.474,13.088,177.4312,0.7183,0.0000
C01305=10.935,-47.018,13.022,176.2893,2.4011,0.0000
C01306=10.132,-46.432,12.887,173.6461,5.1271,0.0000
C01307=9.343,-45.885,12.705,167.0222,8.2576,0.0000
C01308=8.390,-45.503,12.523,156.6479,7.2043,0.0000
C01309=6.990,-45.375,12.387,149.7196,0.2799,0.0000
C01310=4.844,-45.521,12.332,148.3842,-2.4822,0.0000
C01311=2.510,-45.702,12.329,148.2466,-1.7081,0.0000
C01312=0.000,-45.772,12.331,148.2173,0.0003,0.0000
C01313=0.000,-45.772,12.331,148.2173,0.0003,0.0000
C01314=-2.510,-45.702,12.329,148.2466,1.7077,0.0000
C01315=-4.844,-45.521,12.332,148.3843,2.4815,0.0000
C01316=-6.990,-45.375,12.387,149.7196,-0.2794,0.0000
C01317=-8.390,-45.503,12.523,156.6479,-7.2043,0.0000
C01318=-9.343,-45.885,12.705,167.0222,-8.2576,0.0000
C01319=-10.132,-46.432,12.887,173.6461,-5.1271,0.0000
C01320=-10.935,-47.018,13.022,176.2893,-2.4011,0.0000
C01321=-11.930,-47.474,13.088,177.4312,-0.7183,0.0000
C01322=-13.360,-47.661,13.123,179.0290,-0.0208,0.0000
C01323=-15.047,-47.537,13.151,-179.8657,-0.0220,0.0000
C01324=-16.738,-47.094,13.179,179.9573,0.0145,0.0000
C01325=-18.347,-46.510,13.197,179.9960,0.0016,0.0000
C01326=-19.915,-45.860,13.197,179.9960,0.0018,0.0000
C01327=-21.465,-45.136,13.179,179.9596,0.0199,0.0000
C01328=-22.974,-44.253,13.151,-179.8895,-0.0794,0.0000
C01329=-24.255,-43.149,13.123,179.3281,0.7013,0.0000
C01330=-25.133,-42.005,13.088,178.6911,2.3242,0.0000
C01331=-25.514,-40.979,13.022,179.0750,4.3212,0.0000
C01332=-25.668,-39.997,12.887,179.1463,8.1134,0.0000
C01333=-25.839,-39.052,12.705,176.7006,14.9934,0.0000
C01334=-26.243,-38.108,12.523,168.2536,21.5152,0.0000
C01335=-27.143,-37.028,12.387,157.7615,21.0999,0.0000
C01336=-28.763,-35.614,12.332,154.7665,19.8591,0.0000
C01337=-30.541,-34.091,12.329,155.1829,20.5413,0.0000
C01338=-32.366,-32.366,12.331,156.3406,21.8659,0.0000
C01339=-34.091,-30.541,12.329,157.5673,23.1433,0.0000
C01340=-35.614,-28.763,12.332,158.2333,23.6374,0.0000
C01341=-37.028,-27.143,12.387,157.3703,20.6767,0.0000
C01342=-38.108,-26.243,12.523,158.0679,10.9174,0.0000
C01343=-39.052,-25.839,12.705,164.9828,3.1869,0.0000
C01344=-39.997,-25.668,12.887,171.8857,0.8452,0.0000
C01345=-40.979,-25.514,13.022,175.6783,0.9224,0.0000
C01346=-42.005,-25.133,13.088,177.6752,1.3079,0.0000
C01347=-43.149,-24.255,13.123,179.2987,0.6719,0.0000
C01348=-44.253,-22.974,13.151,-179.9206,-0.1105,0.0000
C01349=-45.136,-21.465,13.179,179.9801,0.0404,0.0000
C01350=-45.860,-19.915,13.197,179.9982,0.0040,0.0000
C01351=-46.510,-18.347,13.197,179.9984,0.0040,0.0000
C01352=-47.094,-16.738,13.179,179.9855,0.0427,0.0000
C01353=-47.537,-15.047,13.151,-179.9780,-0.1343,0.0000
C01354=-47.661,-13.360,13.123,-179.9792,0.9710,0.0000
C01355=-47.474,-11.930,13.088,-179.2810,2.5686,0.0000
C01356=-47.018,-10.935,13.022,-177.5938,3.7074,0.0000
C01357=-46.432,-10.132,12.887,-174.8414,6.3283,0.0000
C01358=-45.885,-9.343,12.705,-171.5291,12.8409,0.0000
C01359=-45.503,-8.390,12.523,-172.1606,23.1570,0.0000
C01360=-45.375,-6.990,12.387,-179.6759,30.2800,0.0000
C01361=-45.521,-4.844,12.332,177.0859,31.5827,0.0000
C01362=-45.702,-2.510,12.329,177.9915,31.7377,0.0000
C01363=-45.772,0.000,12.331,-179.9996,31.7827,0.0000
C01364=-45.702,2.510,12.329,-177.9919,31.7377,0.0000
C01365=-45.521,4.844,12.332,-177.0867,31.5827,0.0000
C01366=-45.375,6.990,12.387,179.6765,30.2800,0.0000
C01367=-45.503,8.390,12.523,172.1606,23.1570,0.0000
C01368=-45.885,9.343,12.705,171.5291,12.8409,0.0000
C01369=-46.432,10.132,12.887,174.8414,6.3283,0.0000
C01370=-47.018,10.935,13.022,177.5938,3.7074,0.0000
C01371=-47.474,11.930,13.088,179.2810,2.5686,0.0000
C01372=-47.661,13.360,13.123,179.9792,0.9710,0.0000
C01373=-47.537,15.047,13.151,179.9780,-0.1343,0.0000
C01374=-47.094,16.738,13.179,-179.9855,0.0427,0.0000
C01375=-46.510,18.347,13.197,-179.9984,0.0040,0.0000
C01376=-45.860,19.915,13.197,-179.9982,0.0040,0.0000
C01377=-45.136,21.465,13.179,-179.9801,0.0404,0.0000
C01378=-44.253,22.974,13.151,179.9206,-0.1105,0.0000
C01379=-43.149,24.255,13.123,-179.2987,0.6719,0.0000
C01380=-42.005,25.133,13.088,-177.6752,1.3079,0.0000
C01381=-40.979,25.514,13.022,-175.6783,0.9224,0.0000
C01382=-39.997,25.668,12.887,-171.8857,0.8452,0.0000
C01383=-39.052,25.839,12.705,-164.9828,3.1869,0.0000
C01384=-38.108,26.243,12.523,-158.0679,10.9174,0.0000
C01385=-37.028,27.143,12.387,-157.3700,20.6763,0.0000
C01386=-35.614,28.763,12.332,-158.2337,23.6380,0.0000
C01387=-34.091,30.541,12.329,-157.5676,23.1436,0.0000
C01388=-32.366,32.366,12.331,-156.3402,21.8655,0.0000
C01389=-30.541,34.091,12.329,-155.1831,20.5417,0.0000
C01390=-28.763,35.614,12.332,-154.7670,19.8596,0.0000
C01391=-27.143,37.028,12.387,-157.7612,21.0996,0.0000
C01392=-26.243,38.108,12.523,-168.2536,21.5152,0.0000
C01393=-25.839,39.052,12.705,-176.7006,14.9934,0.0000
C01394=-25.668,39.997,12.887,-179.1463,8.1134,0.0000
C01395=-25.514,40.979,13.022,-179.0750,4.3212,0.0000
C01396=-25.133,42.005,13.088,-178.6911,2.3242,0.0000
C01397=-24.255,43.149,13.123,-179.3281,0.7013,0.0000
C01398=-22.974,44.253,13.151,179.8895,-0.0794,0.0000
C01399=-21.465,45.136,13.179,-179.9596,0.0199,0.0000
C01400=-19.915,45.860,13.197,-179.9960,0.0018,0.0000
C01401=-18.347,46.510,13.197,-179.9960,0.0016,0.0000
C01402=-16.738,47.094,13.179,-179.9573,0.0145,0.0000
C01403=-15.047,47.537,13.151,179.8657,-0.0220,0.0000
C01404=-13.360,47.661,13.123,-179.0290,-0.0208,0.0000
C01405=-11.930,47.474,13.088,-177.4312,-0.7183,0.0000
C01406=-10.935,47.018,13.022,-176.2893,-2.4011,0.0000
C01407=-10.132,46.432,12.887,-173.6461,-5.1271,0.0000
C01408=-9.343,45.885,12.705,-167.0222,-8.2576,0.0000
C01409=-8.390,45.503,12.523,-156.6479,-7.2043,0.0000
C01410=-6.990,45.375,12.387,-149.7196,-0.2794,0.0000
C01411=-4.844,45.521,12.332,-148.3843,2.4815,0.0000
C01412=-2.510,45.702,12.329,-148.2466,1.7077,0.0000
C01413=0.000,45.772,12.331,-148.2173,0.0003,0.0000
C01414=0.000,44.574,14.176,-145.8985,0.0003,0.0000
C01415=2.400,44.508,14.174,-145.9285,-1.8019,0.0000
C01416=4.660,44.338,14.177,-146.0711,-2.3600,0.0000
C01417=6.764,44.232,14.253,-147.8228,1.8796,0.0000
C01418=8.113,44.459,14.440,-158.3173,10.2970,0.0000
C01419=9.024,44.998,14.693,-170.5191,8.6728,0.0000
C01420=9.783,45.750,14.949,-176.4782,4.0286,0.0000
C01421=10.558,46.569,15.143,-178.6653,1.2693,0.0000
C01422=11.519,47.250,15.238,-179.1707,0.3788,0.0000
C01423=12.971,47.615,15.288,-179.8564,0.0153,0.0000
C01424=14.738,47.593,15.328,179.5088,0.0604,0.0000
C01425=16.543,47.159,15.369,-179.9851,-0.0050,0.0000
C01426=18.280,46.536,15.396,-179.9993,-0.0003,0.0000
C01427=19.980,45.832,15.396,-179.9994,-0.0003,0.0000
C01428=21.649,45.044,15.369,-179.9860,-0.0070,0.0000
C01429=23.232,44.075,15.328,179.6100,0.3046,0.0000
C01430=24.496,42.841,15.288,-179.9093,-0.1124,0.0000
C01431=25.266,41.555,15.238,-179.6815,-0.8542,0.0000
C01432=25.464,40.395,15.143,-179.9539,-1.8412,0.0000
C01433=25.432,39.268,14.949,179.6347,-5.3366,0.0000
C01434=25.438,38.199,14.693,-179.4996,-12.8129,0.0000
C01435=25.701,37.174,14.440,-171.8677,-22.5469,0.0000
C01436=26.493,36.060,14.253,-157.3405,-23.5502,0.0000
C01437=28.056,34.647,14.177,-152.9422,-21.4216,0.0000
C01438=29.775,33.169,14.174,-153.2021,-21.9446,0.0000
C01439=31.519,31.519,14.176,-154.4163,-23.3565,0.0000
C01440=33.169,29.775,14.174,-155.7063,-24.7193,0.0000
C01441=34.647,28.056,14.177,-156.2235,-25.0527,0.0000
C01442=36.060,26.493,14.253,-154.7184,-20.6816,0.0000
C01443=37.174,25.701,14.440,-157.2473,-7.5070,0.0000
C01444=38.199,25.438,14.693,-167.1866,-0.4879,0.0000
C01445=39.268,25.432,14.949,-174.6633,0.3637,0.0000
C01446=40.395,25.464,15.143,-178.1587,-0.0460,0.0000
C01447=41.555,25.266,15.238,-179.1457,-0.3185,0.0000
C01448=42.841,24.496,15.288,-179.8876,-0.0907,0.0000
C01449=44.075,23.232,15.328,179.6954,0.3900,0.0000
C01450=45.044,21.649,15.369,-179.9930,-0.0140,0.0000
C01451=45.832,19.980,15.396,-179.9997,-0.0006,0.0000
C01452=46.536,18.280,15.396,-179.9997,-0.0007,0.0000
C01453=47.159,16.543,15.369,-179.9950,-0.0149,0.0000
C01454=47.593,14.738,15.328,179.9396,0.4912,0.0000
C01455=47.615,12.971,15.288,179.9847,-0.1436,0.0000
C01456=47.250,11.519,15.238,179.6212,-0.8293,0.0000
C01457=46.569,10.558,15.143,178.7304,-1.3344,0.0000
C01458=45.750,9.783,14.949,175.9638,-3.5131,0.0000
C01459=44.998,9.024,14.693,171.2089,-9.3715,0.0000
C01460=44.459,8.113,14.440,168.9376,-21.3162,0.0000
C01461=44.232,6.764,14.253,177.7796,-32.1578,0.0000
C01462=44.338,4.660,14.177,-177.1564,-33.8962,0.0000
C01463=44.508,2.400,14.174,-177.8250,-34.0523,0.0000
C01464=44.574,0.000,14.176,179.9996,-34.1015,0.0000
C01465=44.508,-2.400,14.174,177.8255,-34.0523,0.0000
C01466=44.338,-4.660,14.177,177.1575,-33.8961,0.0000
C01467=44.232,-6.764,14.253,-177.7803,-32.1579,0.0000
C01468=44.459,-8.113,14.440,-168.9376,-21.3162,0.0000
C01469=44.998,-9.024,14.693,-171.2089,-9.3715,0.0000
C01470=45.750,-9.783,14.949,-175.9638,-3.5131,0.0000
C01471=46.569,-10.558,15.143,-178.7304,-1.3344,0.0000
C01472=47.250,-11.519,15.238,-179.6212,-0.8293,0.0000
C01473=47.615,-12.971,15.288,-179.9847,-0.1436,0.0000
C01474=47.593,-14.738,15.328,-179.9396,0.4912,0.0000
C01475=47.159,-16.543,15.369,179.9950,-0.0149,0.0000
C01476=46.536,-18.280,15.396,179.9997,-0.0007,0.0000
C01477=45.832,-19.980,15.396,179.9997,-0.0006,0.0000
C01478=45.044,-21.649,15.369,179.9930,-0.0140,0.0000
C01479=44.075,-23.232,15.328,-179.6954,0.3900,0.0000
C01480=42.841,-24.496,15.288,179.8876,-0.0907,0.0000
C01481=41.555,-25.266,15.238,179.1457,-0.3185,0.0000
C01482=40.395,-25.464,15.143,178.1587,-0.0460,0.0000
C01483=39.268,-25.432,14.949,174.6633,0.3637,0.0000
C01484=38.199,-25.438,14.693,167.1866,-0.4879,0.0000
C01485=37.174,-25.701,14.440,157.2473,-7.5070,0.0000
C01486=36.060,-26.493,14.253,154.7181,-20.6811,0.0000
C01487=34.647,-28.056,14.177,156.2241,-25.0535,0.0000
C01488=33.169,-29.775,14.174,155.7066,-24.7197,0.0000
C01489=31.519,-31.519,14.176,154.4159,-23.3560,0.0000
C01490=29.775,-33.169,14.174,153.2024,-21.9449,0.0000
C01491=28.056,-34.647,14.177,152.9429,-21.4223,0.0000
C01492=26.493,-36.060,14.253,157.3400,-23.5498,0.0000
C01493=25.701,-37.174,14.440,171.8677,-22.5469,0.0000
C01494=25.438,-38.199,14.693,179.4996,-12.8129,0.0000
C01495=25.432,-39.268,14.949,-179.6347,-5.3366,0.0000
C01496=25.464,-40.395,15.143,179.9539,-1.8412,0.0000
C01497=25.266,-41.555,15.238,179.6815,-0.8542,0.0000
C01498=24.496,-42.841,15.288,179.9093,-0.1124,0.0000
C01499=23.232,-44.075,15.328,-179.6100,0.3046,0.0000
C01500=21.649,-45.044,15.369,179.9860,-0.0070,0.0000
C01501=19.980,-45.832,15.396,179.9994,-0.0003,0.0000
C01502=18.280,-46.536,15.396,179.9993,-0.0003,0.0000
C01503=16.543,-47.159,15.369,179.9851,-0.0050,0.0000
C01504=14.738,-47.593,15.328,-179.5088,0.0604,0.0000
C01505=12.971,-47.615,15.288,179.8564,0.0153,0.0000
C01506=11.519,-47.250,15.238,179.1707,0.3788,0.0000
C01507=10.558,-46.569,15.143,178.6653,1.2693,0.0000
C01508=9.783,-45.750,14.949,176.4782,4.0286,0.0000
C01509=9.024,-44.998,14.693,170.5191,8.6728,0.0000
C01510=8.113,-44.459,14.440,158.3173,10.2970,0.0000
C01511=6.764,-44.232,14.253,147.8228,1.8796,0.0000
C01512=4.660,-44.338,14.177,146.0711,-2.3600,0.0000
C01513=2.400,-44.508,14.174,145.9285,-1.8019,0.0000
C01514=0.000,-44.574,14.176,145.8985,0.0003,0.0000
C01515=0.000,-44.574,14.176,145.8985,0.0003,0.0000
C01516=-2.400,-44.508,14.174,145.9285,1.8015,0.0000
C01517=-4.660,-44.338,14.177,146.0712,2.3591,0.0000
C01518=-6.764,-44.232,14.253,147.8228,-1.8790,0.0000
C01519=-8.113,-44.459,14.440,158.3173,-10.2970,0.0000
C01520=-9.024,-44.998,14.693,170.5191,-8.6728,0.0000
C01521=-9.783,-45.750,14.949,176.4782,-4.0286,0.0000
C01522=-10.558,-46.569,15.143,178.6653,-1.2693,0.0000
C01523=-11.519,-47.250,15.238,179.1707,-0.3788,0.0000
C01524=-12.971,-47.615,15.288,179.8564,-0.0153,0.0000
C01525=-14.738,-47.593,15.328,-179.5088,-0.0604,0.0000
C01526=-16.543,-47.159,15.369,179.9851,0.0050,0.0000
C01527=-18.280,-46.536,15.396,179.9993,0.0003,0.0000
C01528=-19.980,-45.832,15.396,179.9994,0.0003,0.0000
C01529=-21.649,-45.044,15.369,179.9860,0.0070,0.0000
C01530=-23.232,-44.075,15.328,-179.6100,-0.3046,0.0000
C01531=-24.496,-42.841,15.288,179.9093,0.1124,0.0000
C01532=-25.266,-41.555,15.238,179.6815,0.8542,0.0000
C01533=-25.464,-40.395,15.143,179.9539,1.8412,0.0000
C01534=-25.432,-39.268,14.949,-179.6347,5.3366,0.0000
C01535=-25.438,-38.199,14.693,179.4996,12.8129,0.0000
C01536=-25.701,-37.174,14.440,171.8677,22.5469,0.0000
C01537=-26.493,-36.060,14.253,157.3405,23.5502,0.0000
C01538=-28.056,-34.647,14.177,152.9422,21.4216,0.0000
C01539=-29.775,-33.169,14.174,153.2021,21.9446,0.0000
C01540=-31.519,-31.519,14.176,154.4163,23.3565,0.0000
C01541=-33.169,-29.775,14.174,155.7063,24.7193,0.0000
C01542=-34.647,-28.056,14.177,156.2235,25.0527,0.0000
C01543=-36.060,-26.493,14.253,154.7184,20.6816,0.0000
C01544=-37.174,-25.701,14.440,157.2473,7.5070,0.0000
C01545=-38.199,-25.438,14.693,167.1866,0.4879,0.0000
C01546=-39.268,-25.432,14.949,174.6633,-0.3637,0.0000
C01547=-40.395,-25.464,15.143,178.1587,0.0460,0.0000
C01548=-41.555,-25.266,15.238,179.1457,0.3185,0.0000
C01549=-42.841,-24.496,15.288,179.8876,0.0907,0.0000
C01550=-44.075,-23.232,15.328,-179.6954,-0.3900,0.0000
C01551=-45.044,-21.649,15.369,179.9930,0.0140,0.0000
C01552=-45.832,-19.980,15.396,179.9997,0.0006,0.0000
C01553=-46.536,-18.280,15.396,179.9997,0.0007,0.0000
C01554=-47.159,-16.543,15.369,179.9950,0.0149,0.0000
C01555=-47.593,-14.738,15.328,-179.9396,-0.4912,0.0000
C01556=-47.615,-12.971,15.288,-179.9847,0.1436,0.0000
C01557=-47.250,-11.519,15.238,-179.6212,0.8293,0.0000
C01558=-46.569,-10.558,15.143,-178.7304,1.3344,0.0000
C01559=-45.750,-9.783,14.949,-175.9638,3.5131,0.0000
C01560=-44.998,-9.024,14.693,-171.2089,9.3715,0.0000
C01561=-44.459,-8.113,14.440,-168.9376,21.3162,0.0000
C01562=-44.232,-6.764,14.253,-177.7796,32.1578,0.0000
C01563=-44.338,-4.660,14.177,177.1564,33.8962,0.0000
C01564=-44.508,-2.400,14.174,177.8250,34.0523,0.0000
C01565=-44.574,0.000,14.176,-179.9996,34.1015,0.0000
C01566=-44.508,2.400,14.174,-177.8255,34.0523,0.0000
C01567=-44.338,4.660,14.177,-177.1575,33.8961,0.0000
C01568=-44.232,6.764,14.253,177.7803,32.1579,0.0000
C01569=-44.459,8.113,14.440,168.9376,21.3162,0.0000
C01570=-44.998,9.024,14.693,171.2089,9.3715,0.0000
C01571=-45.750,9.783,14.949,175.9638,3.5131,0.0000
C01572=-46.569,10.558,15.143,178.7304,1.3344,0.0000
C01573=-47.250,11.519,15.238,179.6212,0.8293,0.0000
C01574=-47.615,12.971,15.288,179.9847,0.1436,0.0000
C01575=-47.593,14.738,15.328,179.9396,-0.4912,0.0000
C01576=-47.159,16.543,15.369,-179.9950,0.0149,0.0000
C01577=-46.536,18.280,15.396,-179.9997,0.0007,0.0000
C01578=-45.832,19.980,15.396,-179.9997,0.0006,0.0000
C01579=-45.044,21.649,15.369,-179.9930,0.0140,0.0000
C01580=-44.075,23.232,15.328,179.6954,-0.3900,0.0000
C01581=-42.841,24.496,15.288,-179.8876,0.0907,0.0000
C01582=-41.555,25.266,15.238,-179.1457,0.3185,0.0000
C01583=-40.395,25.464,15.143,-178.1587,0.0460,0.0000
C01584=-39.268,25.432,14.949,-174.6633,-0.3637,0.0000
C01585=-38.199,25.438,14.693,-167.1866,0.4879,0.0000
C01586=-37.174,25.701,14.440,-157.2473,7.5070,0.0000
C01587=-36.060,26.493,14.253,-154.7181,20.6811,0.0000
C01588=-34.647,28.056,14.177,-156.2241,25.0535,0.0000
C01589=-33.169,29.775,14.174,-155.7066,24.7197,0.0000
C01590=-31.519,31.519,14.176,-154.4159,23.3560,0.0000
C01591=-29.775,33.169,14.174,-153.2024,21.9449,0.0000
C01592=-28.056,34.647,14.177,-152.9429,21.4223,0.0000
C01593=-26.493,36.060,14.253,-157.3400,23.5498,0.0000
C01594=-25.701,37.174,14.440,-171.8677,22.5469,0.0000
C01595=-25.438,38.199,14.693,-179.4996,12.8129,0.0000
C01596=-25.432,39.268,14.949,179.6347,5.3366,0.0000
C01597=-25.464,40.395,15.143,-179.9539,1.8412,0.0000
C01598=-25.266,41.555,15.238,-179.6815,0.8542,0.0000
C01599=-24.496,42.841,15.288,-179.9093,0.1124,0.0000
C01600=-23.232,44.075,15.328,179.6100,-0.3046,0.0000
C01601=-21.649,45.044,15.369,-179.9860,0.0070,0.0000
C01602=-19.980,45.832,15.396,-179.9994,0.0003,0.0000
C01603=-18.280,46.536,15.396,-179.9993,0.0003,0.0000
C01604=-16.543,47.159,15.369,-179.9851,0.0050,0.0000
C01605=-14.738,47.593,15.328,179.5088,-0.0604,0.0000
C01606=-12.971,47.615,15.288,-179.8564,-0.0153,0.0000
C01607=-11.519,47.250,15.238,-179.1707,-0.3788,0.0000
C01608=-10.558,46.569,15.143,-178.6653,-1.2693,0.0000
C01609=-9.783,45.750,14.949,-176.4782,-4.0286,0.0000
C01610=-9.024,44.998,14.693,-170.5191,-8.6728,0.0000
C01611=-8.113,44.459,14.440,-158.3173,-10.2970,0.0000
C01612=-6.764,44.232,14.253,-147.8228,-1.8790,0.0000
C01613=-4.660,44.338,14.177,-146.0712,2.3591,0.0000
C01614=-2.400,44.508,14.174,-145.9285,1.8015,0.0000
C01615=0.000,44.574,14.176,-145.8985,0.0003,0.0000
C01616=0.000,43.311,15.978,-144.0999,0.0004,0.0000
C01617=2.285,43.249,15.975,-144.1302,-1.8651,0.0000
C01618=4.466,43.090,15.979,-144.2811,-2.1398,0.0000
C01619=6.526,43.024,16.076,-146.6483,3.7288,0.0000
C01620=7.820,43.354,16.319,-161.4282,12.3849,0.0000
C01621=8.685,44.055,16.652,-173.7915,7.6259,0.0000
C01622=9.411,45.022,16.991,-178.5750,2.1613,0.0000
C01623=10.154,46.088,17.251,179.5618,-0.5669,0.0000
C01624=11.076,47.009,17.379,179.0868,-0.5944,0.0000
C01625=12.553,47.564,17.447,179.2075,-0.1524,0.0000
C01626=14.406,47.654,17.502,179.1191,0.0737,0.0000
C01627=16.332,47.228,17.558,179.9841,0.0052,0.0000
C01628=18.209,46.563,17.595,179.9970,0.0012,0.0000
C01629=20.050,45.800,17.595,179.9971,0.0013,0.0000
C01630=21.847,44.944,17.558,179.9851,0.0076,0.0000
C01631=23.510,43.883,17.502,179.3250,0.5708,0.0000
C01632=24.756,42.510,17.447,179.5473,0.6682,0.0000
C01633=25.408,41.072,17.379,179.7746,1.0660,0.0000
C01634=25.409,39.769,17.251,-179.9089,0.7107,0.0000
C01635=25.181,38.490,16.991,179.4784,-2.5355,0.0000
C01636=25.011,37.293,16.652,178.9511,-9.7663,0.0000
C01637=25.126,36.186,16.319,-175.7805,-21.8159,0.0000
C01638=25.808,35.038,16.076,-157.6953,-25.7162,0.0000
C01639=27.311,33.628,15.979,-151.5865,-22.7136,0.0000
C01640=28.966,32.197,15.975,-151.6440,-23.0225,0.0000
C01641=30.625,30.625,15.978,-152.8941,-24.4962,0.0000
C01642=32.197,28.966,15.975,-154.2248,-25.9199,0.0000
C01643=33.628,27.311,15.979,-154.5487,-26.0347,0.0000
C01644=35.038,25.808,16.076,-152.5004,-19.9959,0.0000
C01645=36.186,25.126,16.319,-158.1304,-3.9168,0.0000
C01646=37.293,25.011,16.652,-170.2321,1.0337,0.0000
C01647=38.490,25.181,16.991,-177.4644,0.5211,0.0000
C01648=39.769,25.409,17.251,179.2893,-0.0911,0.0000
C01649=41.072,25.408,17.379,178.9340,0.2254,0.0000
C01650=42.510,24.756,17.447,179.3318,0.4526,0.0000
C01651=43.883,23.510,17.502,179.4292,0.6749,0.0000
C01652=44.944,21.847,17.558,179.9924,0.0149,0.0000
C01653=45.800,20.050,17.595,179.9987,0.0029,0.0000
C01654=46.563,18.209,17.595,179.9988,0.0030,0.0000
C01655=47.228,16.332,17.558,179.9948,0.0159,0.0000
C01656=47.654,14.406,17.502,179.9263,0.8809,0.0000
C01657=47.564,12.553,17.447,-179.8476,0.7925,0.0000
C01658=47.009,11.076,17.379,-179.4055,0.9131,0.0000
C01659=46.088,10.154,17.251,-179.4331,0.4381,0.0000
C01660=45.022,9.411,16.991,177.8381,-1.4240,0.0000
C01661=44.055,8.685,16.652,172.3297,-6.1533,0.0000
C01662=43.354,7.820,16.319,166.9574,-18.1244,0.0000
C01663=43.024,6.526,16.076,175.5388,-33.2719,0.0000
C01664=43.090,4.466,15.979,-177.3651,-35.6901,0.0000
C01665=43.249,2.285,15.975,-177.6989,-35.8479,0.0000
C01666=43.311,0.000,15.978,179.9996,-35.9001,0.0000
C01667=43.249,-2.285,15.975,177.6995,-35.8479,0.0000
C01668=43.090,-4.466,15.979,177.3664,-35.6901,0.0000
C01669=43.024,-6.526,16.076,-175.5396,-33.2721,0.0000
C01670=43.354,-7.820,16.319,-166.9574,-18.1244,0.0000
C01671=44.055,-8.685,16.652,-172.3297,-6.1533,0.0000
C01672=45.022,-9.411,16.991,-177.8381,-1.4240,0.0000
C01673=46.088,-10.154,17.251,179.4331,0.4381,0.0000
C01674=47.009,-11.076,17.379,179.4055,0.9131,0.0000
C01675=47.564,-12.553,17.447,179.8476,0.7925,0.0000
C01676=47.654,-14.406,17.502,-179.9263,0.8809,0.0000
C01677=47.228,-16.332,17.558,-179.9948,0.0159,0.0000
C01678=46.563,-18.209,17.595,-179.9988,0.0030,0.0000
C01679=45.800,-20.050,17.595,-179.9987,0.0029,0.0000
C01680=44.944,-21.847,17.558,-179.9924,0.0149,0.0000
C01681=43.883,-23.510,17.502,-179.4292,0.6749,0.0000
C01682=42.510,-24.756,17.447,-179.3318,0.4526,0.0000
C01683=41.072,-25.408,17.379,-178.9340,0.2254,0.0000
C01684=39.769,-25.409,17.251,-179.2893,-0.0911,0.0000
C01685=38.490,-25.181,16.991,177.4644,0.5211,0.0000
C01686=37.293,-25.011,16.652,170.2321,1.0337,0.0000
C01687=36.186,-25.126,16.319,158.1304,-3.9168,0.0000
C01688=35.038,-25.808,16.076,152.5001,-19.9952,0.0000
C01689=33.628,-27.311,15.979,154.5493,-26.0356,0.0000
C01690=32.197,-28.966,15.975,154.2251,-25.9202,0.0000
C01691=30.625,-30.625,15.978,152.8936,-24.4957,0.0000
C01692=28.966,-32.197,15.975,151.6443,-23.0229,0.0000
C01693=27.311,-33.628,15.979,151.5873,-22.7144,0.0000
C01694=25.808,-35.038,16.076,157.6946,-25.7158,0.0000
C01695=25.126,-36.186,16.319,175.7805,-21.8159,0.0000
C01696=25.011,-37.293,16.652,-178.9511,-9.7663,0.0000
C01697=25.181,-38.490,16.991,-179.4784,-2.5355,0.0000
C01698=25.409,-39.769,17.251,179.9089,0.7107,0.0000
C01699=25.408,-41.072,17.379,-179.7746,1.0660,0.0000
C01700=24.756,-42.510,17.447,-179.5473,0.6682,0.0000
C01701=23.510,-43.883,17.502,-179.3250,0.5708,0.0000
C01702=21.847,-44.944,17.558,-179.9851,0.0076,0.0000
C01703=20.050,-45.800,17.595,-179.9971,0.0013,0.0000
C01704=18.209,-46.563,17.595,-179.9970,0.0012,0.0000
C01705=16.332,-47.228,17.558,-179.9841,0.0052,0.0000
C01706=14.406,-47.654,17.502,-179.1191,0.0737,0.0000
C01707=12.553,-47.564,17.447,-179.2075,-0.1524,0.0000
C01708=11.076,-47.009,17.379,-179.0868,-0.5944,0.0000
C01709=10.154,-46.088,17.251,-179.5618,-0.5669,0.0000
C01710=9.411,-45.022,16.991,178.5750,2.1613,0.0000
C01711=8.685,-44.055,16.652,173.7915,7.6259,0.0000
C01712=7.820,-43.354,16.319,161.4282,12.3849,0.0000
C01713=6.526,-43.024,16.076,146.6483,3.7288,0.0000
C01714=4.466,-43.090,15.979,144.2811,-2.1398,0.0000
C01715=2.285,-43.249,15.975,144.1302,-1.8651,0.0000
C01716=0.000,-43.311,15.978,144.0999,0.0004,0.0000
C01717=0.000,-43.311,15.978,144.0999,0.0004,0.0000
C01718=-2.285,-43.249,15.975,144.1302,1.8646,0.0000
C01719=-4.466,-43.090,15.979,144.2813,2.1387,0.0000
C01720=-6.526,-43.024,16.076,146.6482,-3.7281,0.0000
C01721=-7.820,-43.354,16.319,161.4282,-12.3849,0.0000
C01722=-8.685,-44.055,16.652,173.7915,-7.6259,0.0000
C01723=-9.411,-45.022,16.991,178.5750,-2.1613,0.0000
C01724=-10.154,-46.088,17.251,-179.5618,0.5669,0.0000
C01725=-11.076,-47.009,17.379,-179.0868,0.5944,0.0000
C01726=-12.553,-47.564,17.447,-179.2075,0.1524,0.0000
C01727=-14.406,-47.654,17.502,-179.1191,-0.0737,0.0000
C01728=-16.332,-47.228,17.558,-179.9841,-0.0052,0.0000
C01729=-18.209,-46.563,17.595,-179.9970,-0.0012,0.0000
C01730=-20.050,-45.800,17.595,-179.9971,-0.0013,0.0000
C01731=-21.847,-44.944,17.558,-179.9851,-0.0076,0.0000
C01732=-23.510,-43.883,17.502,-179.3250,-0.5708,0.0000
C01733=-24.756,-42.510,17.447,-179.5473,-0.6682,0.0000
C01734=-25.408,-41.072,17.379,-179.7746,-1.0660,0.0000
C01735=-25.409,-39.769,17.251,179.9089,-0.7107,0.0000
C01736=-25.181,-38.490,16.991,-179.4784,2.5355,0.0000
C01737=-25.011,-37.293,16.652,-178.9511,9.7663,0.0000
C01738=-25.126,-36.186,16.319,175.7805,21.8159,0.0000
C01739=-25.808,-35.038,16.076,157.6953,25.7162,0.0000
C01740=-27.311,-33.628,15.979,151.5865,22.7136,0.0000
C01741=-28.966,-32.197,15.975,151.6440,23.0225,0.0000
C01742=-30.625,-30.625,15.978,152.8941,24.4962,0.0000
C01743=-32.197,-28.966,15.975,154.2248,25.9199,0.0000
C01744=-33.628,-27.311,15.979,154.5487,26.0347,0.0000
C01745=-35.038,-25.808,16.076,152.5004,19.9959,0.0000
C01746=-36.186,-25.126,16.319,158.1304,3.9168,0.0000
C01747=-37.293,-25.011,16.652,170.2321,-1.0337,0.0000
C01748=-38.490,-25.181,16.991,177.4644,-0.5211,0.0000
C01749=-39.769,-25.409,17.251,-179.2893,0.0911,0.0000
C01750=-41.072,-25.408,17.379,-178.9340,-0.2254,0.0000
C01751=-42.510,-24.756,17.447,-179.3318,-0.4526,0.0000
C01752=-43.883,-23.510,17.502,-179.4292,-0.6749,0.0000
C01753=-44.944,-21.847,17.558,-179.9924,-0.0149,0.0000
C01754=-45.800,-20.050,17.595,-179.9987,-0.0029,0.0000
C01755=-46.563,-18.209,17.595,-179.9988,-0.0030,0.0000
C01756=-47.228,-16.332,17.558,-179.9948,-0.0159,0.0000
C01757=-47.654,-14.406,17.502,-179.9263,-0.8809,0.0000
C01758=-47.564,-12.553,17.447,179.8476,-0.7925,0.0000
C01759=-47.009,-11.076,17.379,179.4055,-0.9131,0.0000
C01760=-46.088,-10.154,17.251,179.4331,-0.4381,0.0000
C01761=-45.022,-9.411,16.991,-177.8381,1.4240,0.0000
C01762=-44.055,-8.685,16.652,-172.3297,6.1533,0.0000
C01763=-43.354,-7.820,16.319,-166.9574,18.1244,0.0000
C01764=-43.024,-6.526,16.076,-175.5388,33.2719,0.0000
C01765=-43.090,-4.466,15.979,177.3651,35.6901,0.0000
C01766=-43.249,-2.285,15.975,177.6989,35.8479,0.0000
C01767=-43.311,0.000,15.978,-179.9996,35.9001,0.0000
C01768=-43.249,2.285,15.975,-177.6995,35.8479,0.0000
C01769=-43.090,4.466,15.979,-177.3664,35.6901,0.0000
C01770=-43.024,6.526,16.076,175.5396,33.2721,0.0000
C01771=-43.354,7.820,16.319,166.9574,18.1244,0.0000
C01772=-44.055,8.685,16.652,172.3297,6.1533,0.0000
C01773=-45.022,9.411,16.991,177.8381,1.4240,0.0000
C01774=-46.088,10.154,17.251,-179.4331,-0.4381,0.0000
C01775=-47.009,11.076,17.379,-179.4055,-0.9131,0.0000
C01776=-47.564,12.553,17.447,-179.8476,-0.7925,0.0000
C01777=-47.654,14.406,17.502,179.9263,-0.8809,0.0000
C01778=-47.228,16.332,17.558,179.9948,-0.0159,0.0000
C01779=-46.563,18.209,17.595,179.9988,-0.0030,0.0000
C01780=-45.800,20.050,17.595,179.9987,-0.0029,0.0000
C01781=-44.944,21.847,17.558,179.9924,-0.0149,0.0000
C01782=-43.883,23.510,17.502,179.4292,-0.6749,0.0000
C01783=-42.510,24.756,17.447,179.3318,-0.4526,0.0000
C01784=-41.072,25.408,17.379,178.9340,-0.2254,0.0000
C01785=-39.769,25.409,17.251,179.2893,0.0911,0.0000
C01786=-38.490,25.181,16.991,-177.4644,-0.5211,0.0000
C01787=-37.293,25.011,16.652,-170.2321,-1.0337,0.0000
C01788=-36.186,25.126,16.319,-158.1304,3.9168,0.0000
C01789=-35.038,25.808,16.076,-152.5001,19.9952,0.0000
C01790=-33.628,27.311,15.979,-154.5493,26.0356,0.0000
C01791=-32.197,28.966,15.975,-154.2251,25.9202,0.0000
C01792=-30.625,30.625,15.978,-152.8936,24.4957,0.0000
C01793=-28.966,32.197,15.975,-151.6443,23.0229,0.0000
C01794=-27.311,33.628,15.979,-151.5873,22.7144,0.0000
C01795=-25.808,35.038,16.076,-157.6946,25.7158,0.0000
C01796=-25.126,36.186,16.319,-175.7805,21.8159,0.0000
C01797=-25.011,37.293,16.652,178.9511,9.7663,0.0000
C01798=-25.181,38.490,16.991,179.4784,2.5355,0.0000
C01799=-25.409,39.769,17.251,-179.9089,-0.7107,0.0000
C01800=-25.408,41.072,17.379,179.7746,-1.0660,0.0000
C01801=-24.756,42.510,17.447,179.5473,-0.6682,0.0000
C01802=-23.510,43.883,17.502,179.3250,-0.5708,0.0000
C01803=-21.847,44.944,17.558,179.9851,-0.0076,0.0000
C01804=-20.050,45.800,17.595,179.9971,-0.0013,0.0000
C01805=-18.209,46.563,17.595,179.9970,-0.0012,0.0000
C01806=-16.332,47.228,17.558,179.9841,-0.0052,0.0000
C01807=-14.406,47.654,17.502,179.1191,-0.0737,0.0000
C01808=-12.553,47.564,17.447,179.2075,0.1524,0.0000
C01809=-11.076,47.009,17.379,179.0868,0.5944,0.0000
C01810=-10.154,46.088,17.251,179.5618,0.5669,0.0000
C01811=-9.411,45.022,16.991,-178.5750,-2.1613,0.0000
C01812=-8.685,44.055,16.652,-173.7915,-7.6259,0.0000
C01813=-7.820,43.354,16.319,-161.4282,-12.3849,0.0000
C01814=-6.526,43.024,16.076,-146.6482,-3.7281,0.0000
C01815=-4.466,43.090,15.979,-144.2813,2.1387,0.0000
C01816=-2.285,43.249,15.975,-144.1302,1.8646,0.0000
C01817=0.000,43.311,15.978,-144.0999,0.0004,0.0000
C01818=0.000,41.999,17.743,-142.7393,0.0003,0.0000
C01819=2.165,41.942,17.740,-142.7694,-1.9027,0.0000
C01820=4.264,41.794,17.745,-142.9344,-1.8367,0.0000
C01821=6.279,41.769,17.866,-146.1515,5.7270,0.0000
C01822=7.515,42.203,18.169,-165.2639,13.0795,0.0000
C01823=8.331,43.070,18.587,-176.3263,5.7834,0.0000
C01824=9.020,44.258,19.017,-179.9189,0.1557,0.0000
C01825=9.729,45.582,19.349,178.4925,-2.5230,0.0000
C01826=10.611,46.755,19.514,177.6906,-1.9837,0.0000
C01827=12.113,47.511,19.602,178.2774,-0.4749,0.0000
C01828=14.056,47.717,19.673,178.7288,0.0593,0.0000
C01829=16.110,47.302,19.746,179.9530,0.0151,0.0000
C01830=18.133,46.592,19.794,179.9934,0.0025,0.0000
C01831=20.124,45.768,19.794,179.9935,0.0029,0.0000
C01832=22.056,44.839,19.746,179.9560,0.0226,0.0000
C01833=23.802,43.680,19.673,179.0591,0.8568,0.0000
C01834=25.030,42.161,19.602,179.1176,1.5538,0.0000
C01835=25.558,40.564,19.514,179.7705,3.0354,0.0000
C01836=25.352,39.110,19.349,-179.2805,2.8495,0.0000
C01837=24.917,37.674,19.017,179.9472,-0.1674,0.0000
C01838=24.565,36.346,18.587,178.4897,-6.6804,0.0000
C01839=24.528,35.156,18.169,-179.0768,-19.5858,0.0000
C01840=25.096,33.975,17.866,-158.7516,-27.5455,0.0000
C01841=26.538,32.569,17.745,-150.6410,-23.7854,0.0000
C01842=28.126,31.188,17.740,-150.4544,-23.8349,0.0000
C01843=29.698,29.698,17.743,-151.7242,-25.3481,0.0000
C01844=31.188,28.126,17.740,-153.0775,-26.8113,0.0000
C01845=32.569,26.538,17.745,-153.1737,-26.6552,0.0000
C01846=33.975,25.096,17.866,-150.7679,-18.7442,0.0000
C01847=35.156,24.528,18.169,-160.4118,-0.8697,0.0000
C01848=36.346,24.565,18.587,-173.3173,1.5000,0.0000
C01849=37.674,24.917,19.017,-179.8326,0.0528,0.0000
C01850=39.110,25.352,19.349,177.1503,-0.7186,0.0000
C01851=40.564,25.558,19.514,176.9646,0.2291,0.0000
C01852=42.161,25.030,19.602,178.4460,0.8821,0.0000
C01853=43.680,23.802,19.673,179.1430,0.9408,0.0000
C01854=44.839,22.056,19.746,179.9774,0.0440,0.0000
C01855=45.768,20.124,19.794,179.9971,0.0065,0.0000
C01856=46.592,18.133,19.794,179.9975,0.0066,0.0000
C01857=47.302,16.110,19.746,179.9849,0.0470,0.0000
C01858=47.717,14.056,19.673,179.9406,1.2712,0.0000
C01859=47.511,12.113,19.602,-179.5249,1.7225,0.0000
C01860=46.755,10.611,19.514,-178.0147,2.3080,0.0000
C01861=45.582,9.729,19.349,-177.4761,1.5061,0.0000
C01862=44.258,9.020,19.017,179.8443,-0.0811,0.0000
C01863=43.070,8.331,18.587,174.2047,-3.6550,0.0000
C01864=42.203,7.515,18.169,166.4917,-14.3455,0.0000
C01865=41.769,6.279,17.866,173.1145,-33.6569,0.0000
C01866=41.794,4.264,17.745,-177.6987,-37.0434,0.0000
C01867=41.942,2.165,17.740,-177.6108,-37.2066,0.0000
C01868=41.999,0.000,17.743,179.9996,-37.2607,0.0000
C01869=41.942,-2.165,17.740,177.6113,-37.2067,0.0000
C01870=41.794,-4.265,17.745,177.7003,-37.0432,0.0000
C01871=41.769,-6.279,17.866,-173.1154,-33.6572,0.0000
C01872=42.203,-7.515,18.169,-166.4917,-14.3455,0.0000
C01873=43.070,-8.331,18.587,-174.2047,-3.6550,0.0000
C01874=44.258,-9.020,19.017,-179.8443,-0.0811,0.0000
C01875=45.582,-9.729,19.349,177.4761,1.5061,0.0000
C01876=46.755,-10.611,19.514,178.0147,2.3080,0.0000
C01877=47.511,-12.113,19.602,179.5249,1.7225,0.0000
C01878=47.717,-14.056,19.673,-179.9406,1.2712,0.0000
C01879=47.302,-16.110,19.746,-179.9849,0.0470,0.0000
C01880=46.592,-18.133,19.794,-179.9975,0.0066,0.0000
C01881=45.768,-20.124,19.794,-179.9971,0.0065,0.0000
C01882=44.839,-22.056,19.746,-179.9774,0.0440,0.0000
C01883=43.680,-23.802,19.673,-179.1430,0.9408,0.0000
C01884=42.161,-25.030,19.602,-178.4460,0.8821,0.0000
C01885=40.564,-25.558,19.514,-176.9646,0.2291,0.0000
C01886=39.110,-25.352,19.349,-177.1503,-0.7186,0.0000
C01887=37.674,-24.917,19.017,179.8326,0.0528,0.0000
C01888=36.346,-24.565,18.587,173.3173,1.5000,0.0000
C01889=35.156,-24.528,18.169,160.4118,-0.8697,0.0000
C01890=33.975,-25.096,17.866,150.7677,-18.7434,0.0000
C01891=32.569,-26.538,17.745,153.1744,-26.6563,0.0000
C01892=31.188,-28.126,17.740,153.0778,-26.8117,0.0000
C01893=29.698,-29.698,17.743,151.7237,-25.3476,0.0000
C01894=28.126,-31.188,17.740,150.4547,-23.8353,0.0000
C01895=26.538,-32.569,17.745,150.6419,-23.7863,0.0000
C01896=25.096,-33.975,17.866,158.7508,-27.5451,0.0000
C01897=24.528,-35.156,18.169,179.0768,-19.5858,0.0000
